KUKA KRL program: MyProgram_307().src

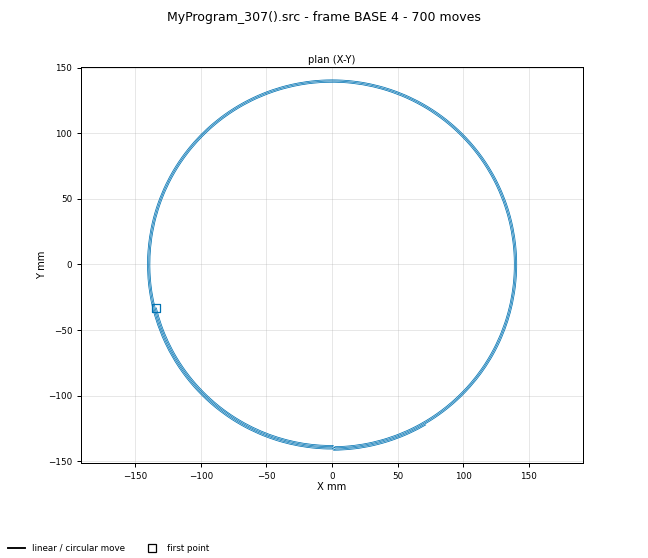
[picture p0: tool path of MyProgram_307().src in frame BASE 4, 700 of 700 moves have a stored position in this frame; points joined in program order, loops and branches not executed]
&ACCESS RVP
&REL 1
&PARAM TEMPLATE = C:\KRC\Roboter\Template\vorgabe
&PARAM EDITMASK = *
DEF MyProgram_307()
; ---- Setting reference (Base) ----
$BASE = BASE_DATA[4]

; --------------------------
; ---- Setting tool (TCP) ----
$TOOL = TOOL_DATA[3]
; --------------------------

$VEL.CP = VEL_APROX_PRINT
Startdeposition()
$VEL.CP = VEL_PRINT
LIN {X -133.9454,Y -33.1389,Z 181,A -162.6013,B 4.9215,C 0.2681,E1 4.7737,E2 255.2334} C_DIS
LIN {X -133.0835,Y -36.4443,Z 181,A -161.1714,B 4.9213,C 0.2719,E1 4.7748,E2 253.8028} C_DIS
LIN {X -132.1601,Y -39.6627,Z 181,A -159.6112,B 4.9212,C 0.2743,E1 4.776,E2 252.2216} C_DIS
LIN {X -131.0021,Y -43.3286,Z 181,A -158.3104,B 4.9208,C 0.281,E1 4.7771,E2 250.9596} C_DIS
LIN {X -130.0909,Y -45.9991,Z 181,A -156.8889,B 4.9208,C 0.2821,E1 4.7784,E2 249.5068} C_DIS
LIN {X -128.9156,Y -49.197,Z 181,A -155.4326,B 4.9206,C 0.2855,E1 4.7799,E2 248.0458} C_DIS
LIN {X -127.6547,Y -52.3816,Z 181,A -153.8465,B 4.9204,C 0.2878,E1 4.7816,E2 246.4393} C_DIS
LIN {X -126.1973,Y -55.7978,Z 181,A -152.4467,B 4.9201,C 0.293,E1 4.7831,E2 245.0586} C_DIS
LIN {X -124.8363,Y -58.7818,Z 181,A -150.8642,B 4.9201,C 0.2946,E1 4.785,E2 243.4483} C_DIS
LIN {X -123.2121,Y -62.1117,Z 181,A -149.5083,B 4.9197,C 0.3,E1 4.7866,E2 242.1167} C_DIS
LIN {X -121.7573,Y -64.9208,Z 181,A -148.0396,B 4.9196,C 0.3019,E1 4.7886,E2 240.6286} C_DIS
LIN {X -120.0477,Y -68.0299,Z 181,A -146.5532,B 4.9194,C 0.3054,E1 4.7906,E2 239.1411} C_DIS
LIN {X -118.3012,Y -71.0238,Z 181,A -144.9881,B 4.9192,C 0.3078,E1 4.7929,E2 237.5603} C_DIS
LIN {X -115.9729,Y -74.7653,Z 181,A -143.1731,B 4.9189,C 0.3122,E1 4.7956,E2 235.7479} C_DIS
LIN {X -113.6464,Y -78.2554,Z 181,A -141.3172,B 4.9188,C 0.3153,E1 4.7985,E2 233.8778} C_DIS
LIN {X -111.4357,Y -81.3732,Z 181,A -139.7753,B 4.9185,C 0.3192,E1 4.801,E2 232.3423} C_DIS
LIN {X -108.9308,Y -84.6964,Z 181,A -137.9766,B 4.9183,C 0.3224,E1 4.8041,E2 230.5349} C_DIS
LIN {X -106.5606,Y -87.6608,Z 181,A -136.3073,B 4.9181,C 0.325,E1 4.807,E2 228.8539} C_DIS
LIN {X -103.6734,Y -91.0571,Z 181,A -134.4884,B 4.9178,C 0.3291,E1 4.8103,E2 227.0397} C_DIS
LIN {X -101.2506,Y -93.7435,Z 181,A -132.8508,B 4.9178,C 0.3309,E1 4.8135,E2 225.3848} C_DIS
LIN {X -98.1988,Y -96.9358,Z 181,A -131.0819,B 4.9174,C 0.3351,E1 4.8169,E2 223.6247} C_DIS
LIN {X -95.6221,Y -99.4784,Z 181,A -129.5752,B 4.9172,C 0.338,E1 4.8199,E2 222.1178} C_DIS
LIN {X -93.0512,Y -101.8874,Z 181,A -127.9603,B 4.9172,C 0.3393,E1 4.8233,E2 220.4833} C_DIS
LIN {X -89.6728,Y -104.8729,Z 181,A -126.0813,B 4.9169,C 0.3425,E1 4.8272,E2 218.6037} C_DIS
LIN {X -86.2779,Y -107.6833,Z 181,A -124.1787,B 4.9168,C 0.345,E1 4.8314,E2 216.6918} C_DIS
LIN {X -82.7629,Y -110.4077,Z 181,A -122.4231,B 4.9165,C 0.3489,E1 4.8352,E2 214.9482} C_DIS
LIN {X -79.8947,Y -112.5007,Z 181,A -120.9123,B 4.9163,C 0.3508,E1 4.8387,E2 213.4328} C_DIS
LIN {X -76.4419,Y -114.8741,Z 181,A -119.086,B 4.9163,C 0.3526,E1 4.8429,E2 211.5952} C_DIS
LIN {X -73.276,Y -116.9196,Z 181,A -117.5586,B 4.916,C 0.3552,E1 4.8465,E2 210.0728} C_DIS
LIN {X -70.2278,Y -118.7753,Z 181,A -115.9776,B 4.916,C 0.3562,E1 4.8503,E2 208.4787} C_DIS
LIN {X -66.4176,Y -120.9472,Z 181,A -114.1055,B 4.9158,C 0.3581,E1 4.8549,E2 206.5998} C_DIS
LIN {X -63.2919,Y -122.6113,Z 181,A -112.7723,B 4.9156,C 0.3612,E1 4.8582,E2 205.2846} C_DIS
LIN {X -60.2633,Y -124.1285,Z 181,A -111.1759,B 4.9156,C 0.3609,E1 4.8622,E2 203.663} C_DIS
LIN {X -56.7836,Y -125.7564,Z 181,A -109.8433,B 4.9153,C 0.3653,E1 4.8655,E2 202.3647} C_DIS
LIN {X -53.8827,Y -127.0278,Z 181,A -108.3761,B 4.9153,C 0.365,E1 4.8694,E2 200.8775} C_DIS
LIN {X -50.3865,Y -128.4531,Z 181,A -106.7907,B 4.9153,C 0.3663,E1 4.8735,E2 199.2895} C_DIS
LIN {X -47.5135,Y -129.5449,Z 181,A -105.5083,B 4.9151,C 0.3674,E1 4.8768,E2 198.0061} C_DIS
LIN {X -44.31,Y -130.6753,Z 181,A -104.1213,B 4.9151,C 0.3688,E1 4.8805,E2 196.6219} C_DIS
LIN {X -41.1844,Y -131.6944,Z 181,A -102.7141,B 4.915,C 0.3694,E1 4.8842,E2 195.2089} C_DIS
LIN {X -37.5841,Y -132.7648,Z 181,A -101.2065,B 4.9149,C 0.3709,E1 4.8883,E2 193.7077} C_DIS
LIN {X -34.6619,Y -133.5589,Z 181,A -99.8819,B 4.9149,C 0.3709,E1 4.8919,E2 192.374} C_DIS
LIN {X -31.53,Y -134.3332,Z 181,A -98.5369,B 4.9149,C 0.3717,E1 4.8955,E2 191.0279} C_DIS
LIN {X -28.3156,Y -135.0474,Z 181,A -97.0137,B 4.9149,C 0.3706,E1 4.8998,E2 189.4836} C_DIS
LIN {X -25.022,Y -135.6957,Z 181,A -95.7674,B 4.9147,C 0.3728,E1 4.9031,E2 188.2564} C_DIS
LIN {X -21.8242,Y -136.2466,Z 181,A -94.4178,B 4.9147,C 0.3732,E1 4.9068,E2 186.9061} C_DIS
LIN {X -18.6385,Y -136.7188,Z 181,A -93.1102,B 4.9147,C 0.3739,E1 4.9104,E2 185.6019} C_DIS
LIN {X -15.2679,Y -137.1353,Z 181,A -91.5885,B 4.9147,C 0.3729,E1 4.9147,E2 184.0648} C_DIS
LIN {X -11.9688,Y -137.4621,Z 181,A -90.4499,B 4.9145,C 0.3758,E1 4.9178,E2 182.9572} C_DIS
LIN {X -9.1803,Y -137.6777,Z 181,A -89.1322,B 4.9146,C 0.3741,E1 4.9215,E2 181.6184} C_DIS
LIN {X -6.0683,Y -137.85,Z 181,A -87.8401,B 4.9146,C 0.3741,E1 4.9251,E2 180.326} C_DIS
LIN {X -3.0627,Y -137.9499,Z 181,A -86.4861,B 4.9147,C 0.3729,E1 4.929,E2 178.9576} C_DIS
LIN {X 0.9801,Y -137.9766,Z 181,A -85.0086,B 4.9146,C 0.375,E1 4.933,E2 177.5057} C_DIS
Enddeposition()
LIN {X 0.9801,Y -137.9766,Z 181,A -85.0086,B 4.9146,C 0.375,E1 4.933,E2 177.5057} C_DIS
Startdeposition()
$VEL.CP = VEL_PRINT
LIN {X 0.4944,Y -138.8836,Z 181,A -85.7347,B 4.875,C 0.383,E1 4.8918,E2 178.3446} C_DIS
LIN {X -3.4627,Y -138.8415,Z 181,A -87.1326,B 4.8752,C 0.3804,E1 4.888,E2 179.7123} C_DIS
LIN {X -6.7652,Y -138.7194,Z 181,A -88.6236,B 4.8752,C 0.3819,E1 4.8838,E2 181.2208} C_DIS
LIN {X -9.6172,Y -138.5516,Z 181,A -89.9061,B 4.875,C 0.383,E1 4.8802,E2 182.5175} C_DIS
LIN {X -13.3672,Y -138.2393,Z 181,A -91.4197,B 4.875,C 0.3824,E1 4.876,E2 184.0265} C_DIS
LIN {X -17.5636,Y -137.7698,Z 181,A -93.0747,B 4.8752,C 0.3811,E1 4.8714,E2 185.6708} C_DIS
LIN {X -21.1736,Y -137.2604,Z 181,A -94.6326,B 4.8752,C 0.3812,E1 4.8671,E2 187.2363} C_DIS
LIN {X -26.796,Y -136.2763,Z 181,A -96.9953,B 4.8752,C 0.3804,E1 4.8606,E2 189.6009} C_DIS
LIN {X -34.4477,Y -134.5442,Z 181,A -100.3956,B 4.8752,C 0.3804,E1 4.8513,E2 193.0236} C_DIS
LIN {X -38.715,Y -133.379,Z 181,A -101.9678,B 4.8755,C 0.3767,E1 4.8471,E2 194.5631} C_DIS
LIN {X -41.235,Y -132.6226,Z 181,A -103.1772,B 4.8755,C 0.3772,E1 4.8439,E2 195.7891} C_DIS
LIN {X -44.9462,Y -131.411,Z 181,A -104.7152,B 4.8756,C 0.3752,E1 4.8398,E2 197.318} C_DIS
LIN {X -48.8191,Y -130.0207,Z 181,A -106.5177,B 4.8756,C 0.3748,E1 4.835,E2 199.1345} C_DIS
LIN {X -51.8681,Y -128.8346,Z 181,A -107.8891,B 4.8757,C 0.3738,E1 4.8315,E2 200.5089} C_DIS
LIN {X -54.7694,Y -127.6288,Z 181,A -109.0264,B 4.8759,C 0.3709,E1 4.8286,E2 201.6256} C_DIS
LIN {X -59.03,Y -125.717,Z 181,A -111.8535,B 4.8754,C 0.3778,E1 4.8211,E2 204.5707} C_DIS
LIN {X -63.9431,Y -123.2899,Z 181,A -113.4971,B 4.8761,C 0.3691,E1 4.8172,E2 206.134} C_DIS
LIN {X -67.9463,Y -121.1302,Z 181,A -115.422,B 4.8762,C 0.3672,E1 4.8125,E2 208.0654} C_DIS
LIN {X -71.7699,Y -118.9046,Z 181,A -117.2904,B 4.8764,C 0.3651,E1 4.808,E2 209.9395} C_DIS
LIN {X -76.6183,Y -115.8401,Z 181,A -119.6162,B 4.8767,C 0.3614,E1 4.8026,E2 212.26} C_DIS
LIN {X -84.2221,Y -110.4349,Z 181,A -123.5852,B 4.877,C 0.3565,E1 4.7935,E2 216.2446} C_DIS
LIN {X -87.516,Y -107.844,Z 181,A -125.375,B 4.8772,C 0.3541,E1 4.7896,E2 218.0422} C_DIS
LIN {X -90.9695,Y -104.9473,Z 181,A -127.3052,B 4.8774,C 0.3515,E1 4.7855,E2 219.9814} C_DIS
LIN {X -94.1981,Y -102.0588,Z 181,A -129.0586,B 4.8776,C 0.3479,E1 4.7819,E2 221.73} C_DIS
LIN {X -97.3086,Y -99.0972,Z 181,A -130.8666,B 4.8779,C 0.3449,E1 4.7782,E2 223.5425} C_DIS
LIN {X -100.4987,Y -95.8605,Z 181,A -132.759,B 4.8781,C 0.3413,E1 4.7745,E2 225.4367} C_DIS
LIN {X -103.3356,Y -92.7954,Z 181,A -134.575,B 4.8783,C 0.3387,E1 4.7711,E2 227.2644} C_DIS
LIN {X -106.3833,Y -89.2849,Z 181,A -136.4902,B 4.8786,C 0.3346,E1 4.7676,E2 229.1787} C_DIS
LIN {X -109.1273,Y -85.9095,Z 181,A -138.2379,B 4.8789,C 0.3304,E1 4.7646,E2 230.9198} C_DIS
LIN {X -111.6331,Y -82.6276,Z 181,A -140.1054,B 4.879,C 0.328,E1 4.7614,E2 232.808} C_DIS
LIN {X -114.241,Y -78.9833,Z 181,A -142.0035,B 4.8793,C 0.3242,E1 4.7583,E2 234.7119} C_DIS
LIN {X -116.2562,Y -75.9861,Z 181,A -143.5562,B 4.8795,C 0.3213,E1 4.7559,E2 236.2723} C_DIS
LIN {X -118.4334,Y -72.5447,Z 181,A -145.232,B 4.8797,C 0.3173,E1 4.7535,E2 237.9468} C_DIS
LIN {X -120.8988,Y -68.358,Z 181,A -147.5502,B 4.8799,C 0.315,E1 4.7502,E2 240.3046} C_DIS
LIN {X -122.5971,Y -65.2626,Z 181,A -148.8178,B 4.8802,C 0.3099,E1 4.7486,E2 241.5473} C_DIS
LIN {X -124.4032,Y -61.7463,Z 181,A -150.4034,B 4.8805,C 0.3055,E1 4.7466,E2 243.1262} C_DIS
LIN {X -125.7912,Y -58.8695,Z 181,A -151.6999,B 4.8807,C 0.302,E1 4.745,E2 244.4194} C_DIS
LIN {X -127.3708,Y -55.3661,Z 181,A -153.2225,B 4.881,C 0.2974,E1 4.7433,E2 245.9331} C_DIS
LIN {X -128.6627,Y -52.2947,Z 181,A -154.5968,B 4.8812,C 0.2938,E1 4.7418,E2 247.3066} C_DIS
LIN {X -129.8975,Y -49.1479,Z 181,A -156.0541,B 4.8814,C 0.2907,E1 4.7403,E2 248.7714} C_DIS
LIN {X -131.4534,Y -44.8238,Z 181,A -158.2954,B 4.8815,C 0.2884,E1 4.7382,E2 251.0561} C_DIS
LIN {X -132.7357,Y -40.8652,Z 181,A -159.9655,B 4.8818,C 0.2834,E1 4.7368,E2 252.7192} C_DIS
LIN {X -133.7465,Y -37.4243,Z 181,A -161.3507,B 4.8821,C 0.2787,E1 4.7357,E2 254.0914} C_DIS
LIN {X -134.4597,Y -34.7807,Z 181,A -162.6813,B 4.8821,C 0.2772,E1 4.7348,E2 255.4472} C_DIS
LIN {X -135.3119,Y -31.2977,Z 181,A -164.1591,B 4.8824,C 0.2731,E1 4.7338,E2 256.9239} C_DIS
LIN {X -135.9929,Y -28.1944,Z 181,A -165.359,B 4.8826,C 0.2686,E1 4.7331,E2 258.1088} C_DIS
LIN {X -136.6755,Y -24.6697,Z 181,A -166.9504,B 4.8828,C 0.2653,E1 4.7323,E2 259.7133} C_DIS
LIN {X -137.2095,Y -21.5023,Z 181,A -168.3304,B 4.883,C 0.2621,E1 4.7317,E2 261.0994} C_DIS
LIN {X -137.6008,Y -18.8473,Z 181,A -169.6654,B 4.883,C 0.2607,E1 4.7312,E2 262.4628} C_DIS
LIN {X -138.0755,Y -14.9645,Z 181,A -171.2559,B 4.8833,C 0.256,E1 4.7306,E2 264.0492} C_DIS
LIN {X -138.4935,Y -10.412,Z 181,A -173.1157,B 4.8836,C 0.2505,E1 4.7302,E2 265.9043} C_DIS
LIN {X -138.7559,Y -5.9941,Z 181,A -175.1528,B 4.8838,C 0.2469,E1 4.7299,E2 267.9671} C_DIS
LIN {X -138.8816,Y -0.8553,Z 181,A -177.5753,B 4.884,C 0.2432,E1 4.7299,E2 270.4261} C_DIS
LIN {X -138.8521,Y 3.0773,Z 181,A -178.8997,B 4.8843,C 0.2363,E1 4.7299,E2 271.7117} C_DIS
LIN {X -138.7439,Y 6.277,Z 181,A 179.7679,B 4.8845,C 0.2327,E1 4.73,E2 273.0446} C_DIS
LIN {X -138.3162,Y 12.5608,Z 181,A 176.8638,B 4.8847,C 0.2276,E1 4.7307,E2 275.9853} C_DIS
LIN {X -137.7408,Y 17.7848,Z 181,A 174.8472,B 4.885,C 0.2204,E1 4.7313,E2 277.9811} C_DIS
LIN {X -137.3589,Y 20.5376,Z 181,A 173.5643,B 4.8851,C 0.2182,E1 4.7318,E2 279.2803} C_DIS
LIN {X -136.7597,Y 24.1988,Z 181,A 172.0031,B 4.8853,C 0.2141,E1 4.7326,E2 280.8441} C_DIS
LIN {X -135.7874,Y 29.1639,Z 181,A 170.1097,B 4.8856,C 0.2068,E1 4.7336,E2 282.7114} C_DIS
LIN {X -135.1804,Y 31.8662,Z 181,A 168.848,B 4.8857,C 0.2046,E1 4.7344,E2 283.9873} C_DIS
LIN {X -134.2777,Y 35.4725,Z 181,A 167.168,B 4.8859,C 0.2015,E1 4.7356,E2 285.6844} C_DIS
LIN {X -133.2631,Y 39.1106,Z 181,A 165.6413,B 4.886,C 0.197,E1 4.7367,E2 287.2058} C_DIS
LIN {X -132.3737,Y 42.0231,Z 181,A 164.275,B 4.8861,C 0.1944,E1 4.7379,E2 288.5848} C_DIS
LIN {X -131.0212,Y 46.0705,Z 181,A 162.3554,B 4.8863,C 0.1909,E1 4.7396,E2 290.523} C_DIS
LIN {X -129.8532,Y 49.2663,Z 181,A 160.5238,B 4.8863,C 0.1905,E1 4.7415,E2 292.4067} C_DIS
LIN {X -128.2055,Y 53.4043,Z 181,A 159.1589,B 4.8866,C 0.182,E1 4.7429,E2 293.7112} C_DIS
LIN {X -126.8991,Y 56.439,Z 181,A 157.8323,B 4.8868,C 0.1782,E1 4.7444,E2 295.0321} C_DIS
LIN {X -125.4412,Y 59.609,Z 181,A 156.2635,B 4.8868,C 0.1755,E1 4.7462,E2 296.6159} C_DIS
LIN {X -124.2073,Y 62.1434,Z 181,A 154.5799,B 4.8868,C 0.1766,E1 4.7484,E2 298.3633} C_DIS
LIN {X -122.152,Y 66.0929,Z 181,A 153.0885,B 4.8871,C 0.1693,E1 4.7503,E2 299.8104} C_DIS
LIN {X -119.9251,Y 70.0521,Z 181,A 151.1744,B 4.8872,C 0.165,E1 4.753,E2 301.7279} C_DIS
LIN {X -117.6653,Y 73.7852,Z 181,A 149.3455,B 4.8874,C 0.1609,E1 4.7557,E2 303.5588} C_DIS
LIN {X -115.2428,Y 77.5143,Z 181,A 147.4169,B 4.8874,C 0.1573,E1 4.7587,E2 305.4975} C_DIS
LIN {X -112.6388,Y 81.2514,Z 181,A 145.5414,B 4.8876,C 0.1529,E1 4.7617,E2 307.3709} C_DIS
LIN {X -109.6966,Y 85.1814,Z 181,A 143.4781,B 4.8877,C 0.1487,E1 4.7652,E2 309.4373} C_DIS
LIN {X -107.1523,Y 88.361,Z 181,A 141.7845,B 4.8879,C 0.1451,E1 4.7682,E2 311.1312} C_DIS
LIN {X -104.6451,Y 91.316,Z 181,A 140.308,B 4.8879,C 0.1407,E1 4.7708,E2 312.5911} C_DIS
LIN {X -102.6132,Y 93.5942,Z 181,A 138.6665,B 4.8879,C 0.1412,E1 4.774,E2 314.279} C_DIS
LIN {X -98.9007,Y 97.5089,Z 181,A 136.5563,B 4.8881,C 0.1358,E1 4.778,E2 316.373} C_DIS
LIN {X -95.8924,Y 100.4682,Z 181,A 134.9128,B 4.8882,C 0.1315,E1 4.7813,E2 318.003} C_DIS
LIN {X -92.6678,Y 103.4499,Z 181,A 132.7945,B 4.8882,C 0.1307,E1 4.7858,E2 320.1578} C_DIS
LIN {X -88.8133,Y 106.7778,Z 181,A 130.7794,B 4.8884,C 0.1262,E1 4.79,E2 322.1606} C_DIS
LIN {X -85.7498,Y 109.2528,Z 181,A 129.1302,B 4.8884,C 0.1235,E1 4.7936,E2 323.8116} C_DIS
LIN {X -82.5228,Y 111.7107,Z 181,A 127.2929,B 4.8884,C 0.1222,E1 4.7978,E2 325.6678} C_DIS
LIN {X -78.2224,Y 114.7635,Z 181,A 125.1824,B 4.8886,C 0.1181,E1 4.8026,E2 327.7686} C_DIS
LIN {X -74.5376,Y 117.1901,Z 181,A 123.3439,B 4.8886,C 0.1156,E1 4.8069,E2 329.6079} C_DIS
LIN {X -70.8603,Y 119.4492,Z 181,A 121.5161,B 4.8886,C 0.1134,E1 4.8113,E2 331.4402} C_DIS
LIN {X -66.8993,Y 121.7123,Z 181,A 119.7049,B 4.8888,C 0.1102,E1 4.8157,E2 333.2412} C_DIS
LIN {X -63.2671,Y 123.6365,Z 181,A 118.1495,B 4.8888,C 0.1068,E1 4.8195,E2 334.7781} C_DIS
LIN {X -61.139,Y 124.7028,Z 181,A 116.618,B 4.8888,C 0.1107,E1 4.8235,E2 336.3765} C_DIS
LIN {X -57.498,Y 126.4254,Z 181,A 115.3336,B 4.8888,C 0.1053,E1 4.8266,E2 337.6135} C_DIS
LIN {X -50.1603,Y 129.5092,Z 181,A 112.0075,B 4.8889,C 0.1023,E1 4.8352,E2 340.9426} C_DIS
LIN {X -46.9783,Y 130.6971,Z 181,A 110.6724,B 4.8889,C 0.1003,E1 4.8387,E2 342.2686} C_DIS
LIN {X -44.2745,Y 131.6382,Z 181,A 109.3595,B 4.8889,C 0.1005,E1 4.8422,E2 343.5971} C_DIS
LIN {X -40.7392,Y 132.7743,Z 181,A 107.8886,B 4.889,C 0.0987,E1 4.8461,E2 345.0594} C_DIS
LIN {X -36.3511,Y 134.0434,Z 181,A 105.8616,B 4.889,C 0.0987,E1 4.8516,E2 347.1029} C_DIS
LIN {X -32.6868,Y 134.9826,Z 181,A 104.5573,B 4.889,C 0.0952,E1 4.8551,E2 348.3746} C_DIS
LIN {X -29.5252,Y 135.7094,Z 181,A 103.2044,B 4.889,C 0.0946,E1 4.8588,E2 349.7285} C_DIS
LIN {X -26.1805,Y 136.394,Z 181,A 101.683,B 4.889,C 0.095,E1 4.863,E2 351.2631} C_DIS
LIN {X -23.3867,Y 136.9018,Z 181,A 100.5739,B 4.8891,C 0.0939,E1 4.866,E2 352.3639} C_DIS
LIN {X -18.7437,Y 137.6151,Z 181,A 98.4444,B 4.8891,C 0.0951,E1 4.8719,E2 354.516} C_DIS
LIN {X -14.9753,Y 138.0743,Z 181,A 96.1048,B 4.8889,C 0.1026,E1 4.8787,E2 356.9492} C_DIS
LIN {X -8.7422,Y 138.6088,Z 181,A 94.3879,B 4.8891,C 0.0933,E1 4.8832,E2 358.5593} C_DIS
LIN {X -5.3578,Y 138.7807,Z 181,A 92.9402,B 4.8891,C 0.0937,E1 4.8872,E2 360.0125} C_DIS
LIN {X -1.1397,Y 138.88,Z 181,A 91.2101,B 4.8891,C 0.0937,E1 4.8921,E2 361.7405} C_DIS
LIN {X 1.7968,Y 138.8735,Z 181,A 90.1301,B 4.8891,C 0.0923,E1 4.895,E2 362.8038} C_DIS
LIN {X 5.3746,Y 138.7801,Z 181,A 88.635,B 4.8891,C 0.0927,E1 4.8992,E2 364.3006} C_DIS
LIN {X 7.8575,Y 138.6633,Z 181,A 87.3994,B 4.8891,C 0.0952,E1 4.9027,E2 365.5618} C_DIS
LIN {X 11.6603,Y 138.3937,Z 181,A 85.9444,B 4.8891,C 0.0944,E1 4.9067,E2 367.0016} C_DIS
LIN {X 15.3454,Y 138.0345,Z 181,A 84.4552,B 4.8891,C 0.0944,E1 4.9109,E2 368.4855} C_DIS
LIN {X 23.4286,Y 136.8948,Z 181,A 81.2082,B 4.8891,C 0.0947,E1 4.9198,E2 371.7167} C_DIS
LIN {X 31.2951,Y 135.3125,Z 181,A 77.7869,B 4.8891,C 0.098,E1 4.9292,E2 375.151} C_DIS
LIN {X 35.2502,Y 134.337,Z 181,A 76.1439,B 4.8891,C 0.0988,E1 4.9336,E2 376.789} C_DIS
LIN {X 38.0632,Y 133.5678,Z 181,A 74.9207,B 4.889,C 0.1001,E1 4.9369,E2 378.0144} C_DIS
LIN {X 41.8152,Y 132.4401,Z 181,A 73.4533,B 4.889,C 0.0997,E1 4.9408,E2 379.463} C_DIS
LIN {X 45.8645,Y 131.0926,Z 181,A 71.5333,B 4.889,C 0.1033,E1 4.9459,E2 381.4025} C_DIS
LIN {X 50.0297,Y 129.56,Z 181,A 69.7647,B 4.8889,C 0.1045,E1 4.9505,E2 383.163} C_DIS
LIN {X 52.8768,Y 128.4258,Z 181,A 68.566,B 4.8889,C 0.1051,E1 4.9536,E2 384.3535} C_DIS
LIN {X 56.2271,Y 126.9938,Z 181,A 67.144,B 4.8889,C 0.1059,E1 4.9572,E2 385.7653} C_DIS
LIN {X 60.9927,Y 124.7749,Z 181,A 64.8954,B 4.8888,C 0.1096,E1 4.963,E2 388.0237} C_DIS
LIN {X 64.6215,Y 122.9337,Z 181,A 63.2427,B 4.8888,C 0.1115,E1 4.967,E2 389.673} C_DIS
LIN {X 68.3111,Y 120.9251,Z 181,A 61.4551,B 4.8887,C 0.1146,E1 4.9714,E2 391.4674} C_DIS
LIN {X 71.9151,Y 118.8168,Z 181,A 59.6705,B 4.8886,C 0.1179,E1 4.9757,E2 393.2596} C_DIS
LIN {X 75.5511,Y 116.5386,Z 181,A 58.1145,B 4.8886,C 0.1181,E1 4.9793,E2 394.7891} C_DIS
LIN {X 81.6596,Y 112.343,Z 181,A 55.002,B 4.8884,C 0.1238,E1 4.9865,E2 397.9087} C_DIS
LIN {X 85.3125,Y 109.595,Z 181,A 53.1419,B 4.8884,C 0.1268,E1 4.9906,E2 399.7658} C_DIS
LIN {X 88.8963,Y 106.7091,Z 181,A 51.2503,B 4.8883,C 0.1302,E1 4.9947,E2 401.6569} C_DIS
LIN {X 92.4054,Y 103.6849,Z 181,A 49.4029,B 4.8882,C 0.133,E1 4.9986,E2 403.4966} C_DIS
LIN {X 95.7081,Y 100.6443,Z 181,A 47.4273,B 4.8881,C 0.1382,E1 5.0026,E2 405.4878} C_DIS
LIN {X 99.4872,Y 96.9106,Z 181,A 45.4732,B 4.8881,C 0.1396,E1 5.0064,E2 407.4128} C_DIS
LIN {X 102.1847,Y 94.0611,Z 181,A 43.8413,B 4.8879,C 0.1432,E1 5.0095,E2 409.0466} C_DIS
LIN {X 105.3046,Y 90.5546,Z 181,A 42.0045,B 4.8879,C 0.146,E1 5.0129,E2 410.8715} C_DIS
LIN {X 107.4021,Y 88.057,Z 181,A 40.562,B 4.8877,C 0.1503,E1 5.0155,E2 412.3266} C_DIS
LIN {X 110.5306,Y 84.097,Z 181,A 38.596,B 4.8877,C 0.1534,E1 5.0188,E2 414.2787} C_DIS
LIN {X 113.1998,Y 80.4683,Z 181,A 36.7609,B 4.8875,C 0.1574,E1 5.0218,E2 416.1114} C_DIS
LIN {X 115.5955,Y 76.9863,Z 181,A 35.0874,B 4.8874,C 0.1606,E1 5.0244,E2 417.7767} C_DIS
LIN {X 117.8647,Y 73.4651,Z 181,A 32.5951,B 4.8869,C 0.175,E1 5.0283,E2 420.3651} C_DIS
LIN {X 121.3088,Y 67.628,Z 181,A 30.6384,B 4.887,C 0.1707,E1 5.0308,E2 422.2182} C_DIS
LIN {X 123.5574,Y 63.4226,Z 181,A 28.9897,B 4.887,C 0.1713,E1 5.0329,E2 423.8274} C_DIS
LIN {X 125.2256,Y 60.0603,Z 181,A 27.1161,B 4.8867,C 0.1797,E1 5.0352,E2 425.7428} C_DIS
LIN {X 127.2538,Y 55.6366,Z 181,A 24.2415,B 4.8861,C 0.1967,E1 5.0386,E2 428.7269} C_DIS
LIN {X 130.3076,Y 48.0531,Z 181,A 21.9685,B 4.8863,C 0.1906,E1 5.0407,E2 430.864} C_DIS
LIN {X 131.6873,Y 44.1272,Z 181,A 20.4175,B 4.8863,C 0.193,E1 5.0421,E2 432.3949} C_DIS
LIN {X 132.7352,Y 40.8669,Z 181,A 19.0565,B 4.8861,C 0.1961,E1 5.0432,E2 433.7501} C_DIS
LIN {X 133.6882,Y 37.6328,Z 181,A 17.7561,B 4.886,C 0.1986,E1 5.0442,E2 435.0397} C_DIS
LIN {X 134.5801,Y 34.3063,Z 181,A 16.3614,B 4.8858,C 0.2022,E1 5.0452,E2 436.432} C_DIS
LIN {X 135.2517,Y 31.5613,Z 181,A 15.0754,B 4.8856,C 0.207,E1 5.046,E2 437.7341} C_DIS
LIN {X 136.5842,Y 25.1796,Z 181,A 12.5906,B 4.8854,C 0.2117,E1 5.0474,E2 440.1945} C_DIS
LIN {X 137.7658,Y 17.5942,Z 181,A 8.9513,B 4.8847,C 0.2272,E1 5.0489,E2 443.8959} C_DIS
LIN {X 138.2931,Y 12.8062,Z 181,A 7.4725,B 4.8848,C 0.2257,E1 5.0493,E2 445.3114} C_DIS
LIN {X 138.5858,Y 9.1154,Z 181,A 6.1341,B 4.8848,C 0.2274,E1 5.0495,E2 446.6267} C_DIS
LIN {X 138.7769,Y 5.4563,Z 181,A 4.5368,B 4.8845,C 0.2329,E1 5.0497,E2 448.2361} C_DIS
LIN {X 138.8787,Y 1.3925,Z 181,A 2.8264,B 4.8842,C 0.2381,E1 5.0498,E2 449.9521} C_DIS
LIN {X 138.8391,Y -3.5486,Z 181,A 1.0016,B 4.8841,C 0.2409,E1 5.0498,E2 451.7509} C_DIS
LIN {X 138.6865,Y -7.4197,Z 181,A -0.641,B 4.8838,C 0.2461,E1 5.0495,E2 453.4004} C_DIS
LIN {X 138.431,Y -11.219,Z 181,A -1.9337,B 4.8838,C 0.2466,E1 5.0493,E2 454.6585} C_DIS
LIN {X 138.0905,Y -14.8251,Z 181,A -3.5008,B 4.8835,C 0.2519,E1 5.0488,E2 456.2362} C_DIS
LIN {X 137.6689,Y -18.3333,Z 181,A -4.728,B 4.8835,C 0.2527,E1 5.0484,E2 457.4347} C_DIS
LIN {X 137.0035,Y -22.7768,Z 181,A -6.6729,B 4.8831,C 0.2593,E1 5.0476,E2 459.3929} C_DIS
LIN {X 136.4329,Y -25.9771,Z 181,A -7.8148,B 4.8831,C 0.2602,E1 5.047,E2 460.5102} C_DIS
LIN {X 135.819,Y -29.0173,Z 181,A -9.3065,B 4.8827,C 0.2668,E1 5.0462,E2 462.0304} C_DIS
LIN {X 135.11,Y -32.1585,Z 181,A -10.6278,B 4.8825,C 0.2704,E1 5.0453,E2 463.3519} C_DIS
LIN {X 133.9712,Y -36.6209,Z 181,A -12.6319,B 4.8822,C 0.2771,E1 5.0439,E2 465.3711} C_DIS
LIN {X 132.384,Y -41.9911,Z 181,A -14.632,B 4.8821,C 0.2791,E1 5.0423,E2 467.3329} C_DIS
LIN {X 131.4752,Y -44.7609,Z 181,A -15.9582,B 4.8818,C 0.2841,E1 5.0411,E2 468.6762} C_DIS
LIN {X 130.0941,Y -48.6232,Z 181,A -17.4787,B 4.8816,C 0.2862,E1 5.0397,E2 470.1758} C_DIS
LIN {X 129.0097,Y -51.4338,Z 181,A -18.7372,B 4.8814,C 0.2898,E1 5.0384,E2 471.4374} C_DIS
LIN {X 127.6641,Y -54.6877,Z 181,A -20.1515,B 4.8812,C 0.2931,E1 5.0369,E2 472.8481} C_DIS
LIN {X 126.1721,Y -58.0459,Z 181,A -21.5854,B 4.8811,C 0.2959,E1 5.0352,E2 474.2725} C_DIS
LIN {X 124.863,Y -60.8141,Z 181,A -22.7598,B 4.8809,C 0.2979,E1 5.0338,E2 475.4366} C_DIS
LIN {X 123.1894,Y -64.1345,Z 181,A -24.3601,B 4.8806,C 0.3028,E1 5.0318,E2 477.0468} C_DIS
LIN {X 121.0072,Y -68.165,Z 181,A -26.2394,B 4.8804,C 0.3074,E1 5.0292,E2 478.9263} C_DIS
LIN {X 118.8168,Y -71.9151,Z 181,A -28.0903,B 4.88,C 0.3127,E1 5.0266,E2 480.7865} C_DIS
LIN {X 116.1817,Y -76.0994,Z 181,A -29.9286,B 4.8799,C 0.3149,E1 5.0238,E2 482.6003} C_DIS
LIN {X 113.8053,Y -79.6095,Z 181,A -31.6792,B 4.8796,C 0.3191,E1 5.0211,E2 484.3526} C_DIS
LIN {X 111.4097,Y -82.9282,Z 181,A -33.1282,B 4.8796,C 0.3198,E1 5.0187,E2 485.7718} C_DIS
LIN {X 109.8516,Y -84.9814,Z 181,A -34.6125,B 4.879,C 0.328,E1 5.0161,E2 487.312} C_DIS
LIN {X 107.6277,Y -87.7809,Z 181,A -35.6175,B 4.8792,C 0.3249,E1 5.0145,E2 488.2569} C_DIS
LIN {X 105.6543,Y -90.1468,Z 181,A -37.0951,B 4.8788,C 0.3306,E1 5.0117,E2 489.7627} C_DIS
LIN {X 102.6332,Y -93.572,Z 181,A -39.1631,B 4.8784,C 0.3372,E1 5.0078,E2 491.8563} C_DIS
LIN {X 100.0797,Y -96.2987,Z 181,A -40.4539,B 4.8784,C 0.3371,E1 5.0054,E2 493.1157} C_DIS
LIN {X 96.8246,Y -99.5705,Z 181,A -42.3048,B 4.8782,C 0.3403,E1 5.0017,E2 494.9613} C_DIS
LIN {X 93.5242,Y -102.6766,Z 181,A -44.0905,B 4.878,C 0.3429,E1 4.9981,E2 496.7376} C_DIS
LIN {X 91.0189,Y -104.9043,Z 181,A -45.5269,B 4.8778,C 0.3464,E1 4.9951,E2 498.1822} C_DIS
LIN {X 87.3953,Y -107.9413,Z 181,A -47.1761,B 4.8778,C 0.3461,E1 4.9916,E2 499.7934} C_DIS
LIN {X 83.4862,Y -110.9918,Z 181,A -49.2192,B 4.8775,C 0.3498,E1 4.9871,E2 501.8379} C_DIS
LIN {X 79.4002,Y -113.951,Z 181,A -51.4179,B 4.8771,C 0.3549,E1 4.982,E2 504.0538} C_DIS
LIN {X 75.7087,Y -116.4362,Z 181,A -53.2184,B 4.8769,C 0.3575,E1 4.9778,E2 505.8511} C_DIS
LIN {X 71.9893,Y -118.7719,Z 181,A -55.1148,B 4.8767,C 0.3615,E1 4.9733,E2 507.7601} C_DIS
LIN {X 66.8547,Y -121.7366,Z 181,A -57.4074,B 4.8765,C 0.3632,E1 4.9678,E2 510.0344} C_DIS
LIN {X 63.578,Y -123.4782,Z 181,A -58.7569,B 4.8765,C 0.3631,E1 4.9645,E2 511.3611} C_DIS
LIN {X 60.2279,Y -125.1455,Z 181,A -60.3713,B 4.8763,C 0.3661,E1 4.9604,E2 512.986} C_DIS
LIN {X 56.9719,Y -126.6607,Z 181,A -61.8128,B 4.8763,C 0.3675,E1 4.9568,E2 514.4233} C_DIS
LIN {X 53.8374,Y -128.0246,Z 181,A -63.2161,B 4.8761,C 0.3691,E1 4.9532,E2 515.8267} C_DIS
LIN {X 50.6593,Y -129.3153,Z 181,A -64.5977,B 4.876,C 0.3704,E1 4.9496,E2 517.2049} C_DIS
LIN {X 47.8314,Y -130.3895,Z 181,A -65.9959,B 4.8757,C 0.3736,E1 4.9459,E2 518.6238} C_DIS
LIN {X 44.2597,Y -131.6432,Z 181,A -67.4206,B 4.8757,C 0.3736,E1 4.9422,E2 520.0315} C_DIS
LIN {X 41.2504,Y -132.6179,Z 181,A -68.5997,B 4.8757,C 0.3733,E1 4.9391,E2 521.195} C_DIS
LIN {X 37.4427,Y -133.7413,Z 181,A -70.0701,B 4.8758,C 0.3727,E1 4.9352,E2 522.6442} C_DIS
LIN {X 34.2504,Y -134.5943,Z 181,A -71.9656,B 4.8752,C 0.3803,E1 4.9299,E2 524.6109} C_DIS
LIN {X 30.91,Y -135.4005,Z 181,A -73.0582,B 4.8754,C 0.3775,E1 4.927,E2 525.6616} C_DIS
LIN {X 27.7361,Y -136.0861,Z 181,A -74.3672,B 4.8754,C 0.3781,E1 4.9234,E2 526.9673} C_DIS
LIN {X 23.3692,Y -136.9047,Z 181,A -76.0893,B 4.8754,C 0.3779,E1 4.9187,E2 528.6759} C_DIS
LIN {X 17.0841,Y -137.8307,Z 181,A -78.9059,B 4.8751,C 0.3816,E1 4.9109,E2 531.5199} C_DIS
LIN {X 13.2866,Y -138.247,Z 181,A -80.3758,B 4.8751,C 0.3811,E1 4.9068,E2 532.9767} C_DIS
LIN {X 9.6364,Y -138.5502,Z 181,A -81.8724,B 4.8751,C 0.3814,E1 4.9026,E2 534.4722} C_DIS
LIN {X 5.8085,Y -138.7632,Z 181,A -83.434,B 4.8751,C 0.3816,E1 4.8983,E2 536.032} C_DIS
LIN {X 2.3643,Y -138.864,Z 181,A -84.9097,B 4.8751,C 0.3825,E1 4.8941,E2 537.5155} C_DIS
LIN {X 2.3643,Y -138.864,Z 181,A -84.9097,B 4.8751,C 0.3825,E1 4.8941,E2 537.5155} C_DIS
Enddeposition()
LIN {X 0.998,Y -139.78,Z 181,A -84.9749,B 4.8345,C 0.3788,E1 4.8533,E2 537.5584} C_DIS
Startdeposition()
$VEL.CP = VEL_PRINT
LIN {X 4.0371,Y -139.7283,Z 181,A -83.5714,B 4.8346,C 0.3767,E1 4.8572,E2 536.1332} C_DIS
LIN {X 7.3998,Y -139.591,Z 181,A -82.163,B 4.8346,C 0.376,E1 4.8612,E2 534.7203} C_DIS
LIN {X 11.0635,Y -139.3497,Z 181,A -80.5381,B 4.8348,C 0.3741,E1 4.8658,E2 533.0784} C_DIS
LIN {X 14.9873,Y -138.9806,Z 181,A -79.0366,B 4.8348,C 0.3748,E1 4.8699,E2 531.5913} C_DIS
LIN {X 19.0382,Y -138.4856,Z 181,A -77.0101,B 4.8352,C 0.3698,E1 4.8756,E2 529.5162} C_DIS
LIN {X 22.7089,Y -137.9297,Z 181,A -76.0761,B 4.8347,C 0.3759,E1 4.878,E2 528.6605} C_DIS
LIN {X 28.1751,Y -136.9177,Z 181,A -74.0311,B 4.8346,C 0.3773,E1 4.8836,E2 526.6455} C_DIS
LIN {X 31.0752,Y -136.2883,Z 181,A -71.95,B 4.8355,C 0.3659,E1 4.8895,E2 524.4473} C_DIS
LIN {X 35.3263,Y -135.2506,Z 181,A -70.5785,B 4.8352,C 0.3696,E1 4.8931,E2 523.1318} C_DIS
LIN {X 40.0072,Y -133.9408,Z 181,A -68.6784,B 4.8352,C 0.3689,E1 4.8982,E2 521.2429} C_DIS
LIN {X 42.7538,Y -133.0876,Z 181,A -67.4647,B 4.8354,C 0.3673,E1 4.9014,E2 520.0236} C_DIS
LIN {X 46.2041,Y -131.9299,Z 181,A -65.9853,B 4.8354,C 0.3659,E1 4.9053,E2 518.5449} C_DIS
LIN {X 49.7703,Y -130.628,Z 181,A -64.33,B 4.8357,C 0.3629,E1 4.9097,E2 516.8751} C_DIS
LIN {X 53.8319,Y -129.0048,Z 181,A -62.6406,B 4.8357,C 0.3621,E1 4.914,E2 515.1983} C_DIS
LIN {X 57.2773,Y -127.5126,Z 181,A -61.1762,B 4.8358,C 0.3611,E1 4.9177,E2 513.7429} C_DIS
LIN {X 60.4029,Y -126.062,Z 181,A -59.7691,B 4.836,C 0.3593,E1 4.9213,E2 512.3354} C_DIS
LIN {X 63.5714,Y -124.4942,Z 181,A -58.3184,B 4.8361,C 0.3573,E1 4.9249,E2 510.8833} C_DIS
LIN {X 67.2431,Y -122.5527,Z 181,A -56.0459,B 4.8368,C 0.3474,E1 4.9307,E2 508.5326} C_DIS
LIN {X 71.8447,Y -119.9129,Z 181,A -54.694,B 4.8363,C 0.3548,E1 4.9337,E2 507.29} C_DIS
LIN {X 76.0217,Y -117.3089,Z 181,A -52.6076,B 4.8366,C 0.3506,E1 4.9386,E2 505.1928} C_DIS
LIN {X 79.3106,Y -115.1111,Z 181,A -50.6096,B 4.8371,C 0.3429,E1 4.9434,E2 503.1429} C_DIS
LIN {X 82.364,Y -112.9467,Z 181,A -49.4544,B 4.837,C 0.3452,E1 4.9459,E2 502.0375} C_DIS
LIN {X 85.7552,Y -110.3936,Z 181,A -47.6526,B 4.8373,C 0.3413,E1 4.9499,E2 500.2259} C_DIS
LIN {X 89.1806,Y -107.6452,Z 181,A -45.8695,B 4.8375,C 0.3381,E1 4.9537,E2 498.4435} C_DIS
LIN {X 92.0347,Y -105.2156,Z 181,A -44.4193,B 4.8376,C 0.3363,E1 4.9568,E2 497.0036} C_DIS
LIN {X 95.2741,Y -102.2913,Z 181,A -42.6315,B 4.8379,C 0.3327,E1 4.9605,E2 495.2145} C_DIS
LIN {X 98.6584,Y -99.0314,Z 181,A -40.7627,B 4.8381,C 0.3295,E1 4.9642,E2 493.3517} C_DIS
LIN {X 101.7542,Y -95.8476,Z 181,A -39.1497,B 4.8381,C 0.3285,E1 4.9672,E2 491.7647} C_DIS
LIN {X 104.8141,Y -92.4916,Z 181,A -37.244,B 4.8385,C 0.3238,E1 4.9708,E2 489.8516} C_DIS
LIN {X 107.3241,Y -89.5675,Z 181,A -35.6059,B 4.8387,C 0.3195,E1 4.9738,E2 488.2043} C_DIS
LIN {X 112.2788,Y -83.2719,Z 181,A -32.6403,B 4.839,C 0.3163,E1 4.9788,E2 485.2784} C_DIS
LIN {X 114.026,Y -80.8632,Z 181,A -31.4278,B 4.8391,C 0.3136,E1 4.9808,E2 484.0659} C_DIS
LIN {X 115.9162,Y -78.1293,Z 181,A -29.872,B 4.8395,C 0.3076,E1 4.9833,E2 482.483} C_DIS
LIN {X 119.6744,Y -72.2407,Z 181,A -27.1201,B 4.8399,C 0.3021,E1 4.9874,E2 479.7436} C_DIS
LIN {X 121.7339,Y -68.7138,Z 181,A -25.4328,B 4.8401,C 0.2978,E1 4.9897,E2 478.053} C_DIS
LIN {X 123.81,Y -64.8937,Z 181,A -23.7704,B 4.8403,C 0.2949,E1 4.9919,E2 476.4049} C_DIS
LIN {X 125.6096,Y -61.3405,Z 181,A -22.2333,B 4.8405,C 0.292,E1 4.9938,E2 474.8791} C_DIS
LIN {X 126.9674,Y -58.4759,Z 181,A -20.9397,B 4.8407,C 0.2887,E1 4.9953,E2 473.5852} C_DIS
LIN {X 128.4557,Y -55.1306,Z 181,A -19.4651,B 4.8409,C 0.2851,E1 4.9969,E2 472.1127} C_DIS
LIN {X 129.7721,Y -51.9562,Z 181,A -18.1433,B 4.841,C 0.2826,E1 4.9983,E2 470.8012} C_DIS
LIN {X 130.9402,Y -48.9368,Z 181,A -16.8021,B 4.8413,C 0.2788,E1 4.9996,E2 469.457} C_DIS
LIN {X 132.1026,Y -45.706,Z 181,A -15.4003,B 4.8415,C 0.2751,E1 5.0009,E2 468.0547} C_DIS
LIN {X 133.2118,Y -42.3651,Z 181,A -13.4173,B 4.8421,C 0.2635,E1 5.0027,E2 465.9987} C_DIS
LIN {X 134.7611,Y -37.1466,Z 181,A -11.9506,B 4.8418,C 0.2683,E1 5.0037,E2 464.6317} C_DIS
LIN {X 135.9013,Y -32.7261,Z 181,A -10.0545,B 4.8422,C 0.2627,E1 5.005,E2 462.7308} C_DIS
LIN {X 136.7045,Y -29.192,Z 181,A -8.5998,B 4.8424,C 0.259,E1 5.0059,E2 461.2789} C_DIS
LIN {X 137.971,Y -22.4616,Z 181,A -5.931,B 4.8427,C 0.2531,E1 5.0072,E2 458.6262} C_DIS
LIN {X 138.3457,Y -20.0182,Z 181,A -4.9156,B 4.8428,C 0.2502,E1 5.0076,E2 457.6096} C_DIS
LIN {X 138.827,Y -16.3503,Z 181,A -3.4586,B 4.843,C 0.2468,E1 5.0081,E2 456.1593} C_DIS
LIN {X 139.2039,Y -12.7615,Z 181,A -2.0099,B 4.8432,C 0.243,E1 5.0085,E2 454.7135} C_DIS
LIN {X 139.5171,Y -8.6743,Z 181,A -0.3108,B 4.8434,C 0.238,E1 5.0088,E2 453.0106} C_DIS
LIN {X 139.7249,Y -4.1566,Z 181,A 1.4575,B 4.8436,C 0.2339,E1 5.009,E2 451.2521} C_DIS
LIN {X 139.7866,Y -0.3566,Z 181,A 3.0491,B 4.8439,C 0.229,E1 5.009,E2 449.6549} C_DIS
LIN {X 139.7315,Y 3.9212,Z 181,A 4.6513,B 4.8439,C 0.2262,E1 5.009,E2 448.0713} C_DIS
LIN {X 139.5721,Y 7.775,Z 181,A 6.3037,B 4.8442,C 0.2207,E1 5.0087,E2 446.4085} C_DIS
LIN {X 139.2873,Y 11.8023,Z 181,A 7.7617,B 4.8443,C 0.2188,E1 5.0084,E2 444.9749} C_DIS
LIN {X 138.9409,Y 15.3559,Z 181,A 9.3083,B 4.8446,C 0.2135,E1 5.008,E2 443.4165} C_DIS
LIN {X 137.8278,Y 23.3194,Z 181,A 11.9915,B 4.8446,C 0.2129,E1 5.007,E2 440.8109} C_DIS
LIN {X 136.9118,Y 28.2038,Z 181,A 14.5414,B 4.8451,C 0.2,E1 5.0056,E2 438.1931} C_DIS
LIN {X 136.0741,Y 32.0092,Z 181,A 15.9053,B 4.8451,C 0.1988,E1 5.0047,E2 436.8587} C_DIS
LIN {X 134.9382,Y 36.4979,Z 181,A 17.7483,B 4.8454,C 0.1944,E1 5.0035,E2 435.0216} C_DIS
LIN {X 134.0855,Y 39.5131,Z 181,A 19.0507,B 4.8455,C 0.1906,E1 5.0024,E2 433.7162} C_DIS
LIN {X 133.077,Y 42.7868,Z 181,A 20.4016,B 4.8456,C 0.1876,E1 5.0013,E2 432.3713} C_DIS
LIN {X 131.9647,Y 46.1038,Z 181,A 21.8349,B 4.8458,C 0.1837,E1 5,E2 430.9374} C_DIS
LIN {X 130.1008,Y 51.1275,Z 181,A 24.3727,B 4.8462,C 0.1731,E1 4.9974,E2 428.3541} C_DIS
LIN {X 128.4815,Y 55.0711,Z 181,A 25.4812,B 4.846,C 0.1774,E1 4.9963,E2 427.3275} C_DIS
LIN {X 126.7172,Y 59.017,Z 181,A 27.3705,B 4.8462,C 0.1712,E1 4.9941,E2 425.4222} C_DIS
LIN {X 125.1202,Y 62.3324,Z 181,A 28.8465,B 4.8464,C 0.1678,E1 4.9923,E2 423.9497} C_DIS
LIN {X 123.3489,Y 65.7716,Z 181,A 30.4993,B 4.8465,C 0.1629,E1 4.9901,E2 422.2876} C_DIS
LIN {X 120.9205,Y 70.134,Z 181,A 32.7669,B 4.8468,C 0.1548,E1 4.987,E2 419.9905} C_DIS
LIN {X 118.8345,Y 73.6146,Z 181,A 34.1017,B 4.8468,C 0.1553,E1 4.9851,E2 418.6976} C_DIS
LIN {X 116.3686,Y 77.4536,Z 181,A 35.9205,B 4.8468,C 0.1515,E1 4.9823,E2 416.8847} C_DIS
LIN {X 113.7843,Y 81.2024,Z 181,A 37.731,B 4.847,C 0.1479,E1 4.9794,E2 415.0807} C_DIS
LIN {X 111.1865,Y 84.7247,Z 181,A 39.501,B 4.8471,C 0.1441,E1 4.9764,E2 413.3132} C_DIS
LIN {X 107.1261,Y 89.8035,Z 181,A 41.983,B 4.8472,C 0.1406,E1 4.9721,E2 410.8539} C_DIS
LIN {X 104.6579,Y 92.6683,Z 181,A 43.5992,B 4.8473,C 0.1364,E1 4.9691,E2 409.2289} C_DIS
LIN {X 101.5104,Y 96.106,Z 181,A 45.4636,B 4.8474,C 0.133,E1 4.9656,E2 407.37} C_DIS
LIN {X 98.358,Y 99.3299,Z 181,A 47.8158,B 4.8477,C 0.1227,E1 4.9608,E2 404.9527} C_DIS
LIN {X 94.5408,Y 102.9695,Z 181,A 49.2528,B 4.8476,C 0.1279,E1 4.958,E2 403.6082} C_DIS
LIN {X 91.7699,Y 105.4466,Z 181,A 50.8668,B 4.8476,C 0.1238,E1 4.9546,E2 401.9824} C_DIS
LIN {X 88.1697,Y 108.4754,Z 181,A 52.7603,B 4.8478,C 0.1207,E1 4.9506,E2 400.0932} C_DIS
LIN {X 84.6719,Y 111.2269,Z 181,A 54.5717,B 4.8478,C 0.1177,E1 4.9466,E2 398.2833} C_DIS
LIN {X 80.855,Y 114.0318,Z 181,A 56.702,B 4.848,C 0.112,E1 4.9417,E2 396.1288} C_DIS
LIN {X 77.9666,Y 116.0261,Z 181,A 57.6424,B 4.8479,C 0.1159,E1 4.9397,E2 395.2517} C_DIS
LIN {X 73.7547,Y 118.7473,Z 181,A 59.9274,B 4.848,C 0.1098,E1 4.9342,E2 392.9374} C_DIS
LIN {X 69.8074,Y 121.1101,Z 181,A 61.7479,B 4.848,C 0.1079,E1 4.9298,E2 391.1253} C_DIS
LIN {X 65.8663,Y 123.2981,Z 181,A 63.7644,B 4.8482,C 0.1032,E1 4.9248,E2 389.0875} C_DIS
LIN {X 61.6384,Y 125.4626,Z 181,A 65.6772,B 4.8482,C 0.1011,E1 4.9201,E2 387.179} C_DIS
LIN {X 56.7647,Y 127.7419,Z 181,A 67.5827,B 4.8482,C 0.102,E1 4.9153,E2 385.3118} C_DIS
LIN {X 53.7728,Y 129.0295,Z 181,A 68.9692,B 4.8482,C 0.0999,E1 4.9117,E2 383.919} C_DIS
LIN {X 49.921,Y 130.5704,Z 181,A 70.5953,B 4.8482,C 0.0989,E1 4.9075,E2 382.3026} C_DIS
LIN {X 46.2951,Y 131.8984,Z 181,A 72.7007,B 4.8484,C 0.0911,E1 4.9018,E2 380.131} C_DIS
LIN {X 41.7591,Y 133.4053,Z 181,A 74.0915,B 4.8484,C 0.0961,E1 4.8983,E2 378.8128} C_DIS
LIN {X 37.117,Y 134.7694,Z 181,A 76.026,B 4.8484,C 0.095,E1 4.8931,E2 376.8848} C_DIS
LIN {X 34.2378,Y 135.5285,Z 181,A 77.5621,B 4.8484,C 0.0904,E1 4.8889,E2 375.3091} C_DIS
LIN {X 31.0601,Y 136.2918,Z 181,A 78.9382,B 4.8484,C 0.0891,E1 4.8851,E2 373.9287} C_DIS
LIN {X 27.5876,Y 137.0372,Z 181,A 80.0795,B 4.8484,C 0.0918,E1 4.8821,E2 372.8277} C_DIS
LIN {X 23.4052,Y 137.8135,Z 181,A 82.1084,B 4.8484,C 0.0876,E1 4.8764,E2 370.7633} C_DIS
LIN {X 20.0062,Y 138.3475,Z 181,A 83.2845,B 4.8484,C 0.0896,E1 4.8732,E2 369.6172} C_DIS
LIN {X 15.9034,Y 138.8803,Z 181,A 84.8577,B 4.8484,C 0.0902,E1 4.8689,E2 368.0601} C_DIS
LIN {X 12.805,Y 139.1998,Z 181,A 86.1364,B 4.8484,C 0.0898,E1 4.8654,E2 366.7816} C_DIS
LIN {X 9.5678,Y 139.4599,Z 181,A 87.5791,B 4.8484,C 0.0882,E1 4.8613,E2 365.3254} C_DIS
LIN {X 5.5594,Y 139.6759,Z 181,A 89.1355,B 4.8484,C 0.0889,E1 4.857,E2 363.7808} C_DIS
LIN {X 1.9899,Y 139.7727,Z 181,A 90.5628,B 4.8484,C 0.0891,E1 4.853,E2 362.3587} C_DIS
LIN {X -1.968,Y 139.7731,Z 181,A 92.2589,B 4.8484,C 0.0883,E1 4.8483,E2 360.654} C_DIS
LIN {X -5.7313,Y 139.6692,Z 181,A 93.765,B 4.8484,C 0.0887,E1 4.8441,E2 359.1533} C_DIS
LIN {X -10.2185,Y 139.4124,Z 181,A 95.9853,B 4.8485,C 0.085,E1 4.8377,E2 356.8861} C_DIS
LIN {X -14.1892,Y 139.0664,Z 181,A 97.2003,B 4.8485,C 0.0897,E1 4.8345,E2 355.7249} C_DIS
LIN {X -19.2498,Y 138.4555,Z 181,A 100.1179,B 4.8485,C 0.0818,E1 4.8262,E2 352.7035} C_DIS
LIN {X -25.2061,Y 137.4962,Z 181,A 101.6145,B 4.8484,C 0.0929,E1 4.8224,E2 351.3318} C_DIS
LIN {X -29.4035,Y 136.6588,Z 181,A 103.634,B 4.8484,C 0.0911,E1 4.8168,E2 349.28} C_DIS
LIN {X -32.7698,Y 135.8908,Z 181,A 104.9928,B 4.8484,C 0.0925,E1 4.8131,E2 347.9292} C_DIS
LIN {X -36.2597,Y 135.0017,Z 181,A 106.5456,B 4.8484,C 0.0928,E1 4.8089,E2 346.3676} C_DIS
LIN {X -41.126,Y 133.5996,Z 181,A 108.5677,B 4.8484,C 0.0949,E1 4.8035,E2 344.3535} C_DIS
LIN {X -44.5768,Y 132.4886,Z 181,A 110.0707,B 4.8484,C 0.0959,E1 4.7995,E2 342.8493} C_DIS
LIN {X -47.6773,Y 131.4043,Z 181,A 111.4782,B 4.8483,C 0.0966,E1 4.7958,E2 341.435} C_DIS
LIN {X -52.0437,Y 129.7368,Z 181,A 113.7171,B 4.8483,C 0.0954,E1 4.7898,E2 339.1566} C_DIS
LIN {X -55.3264,Y 128.371,Z 181,A 114.5939,B 4.8482,C 0.1024,E1 4.7878,E2 338.3539} C_DIS
LIN {X -58.1282,Y 127.1282,Z 181,A 116.3143,B 4.8482,C 0.0995,E1 4.7832,E2 336.5762} C_DIS
LIN {X -62.0146,Y 125.277,Z 181,A 117.9515,B 4.8482,C 0.1028,E1 4.7792,E2 334.9562} C_DIS
LIN {X -64.9517,Y 123.7795,Z 181,A 119.2588,B 4.8482,C 0.1049,E1 4.7759,E2 333.6554} C_DIS
LIN {X -68.7184,Y 121.7313,Z 181,A 121.1664,B 4.8482,C 0.1059,E1 4.7712,E2 331.7303} C_DIS
LIN {X -72.1109,Y 119.7529,Z 181,A 122.6494,B 4.848,C 0.1093,E1 4.7677,E2 330.2644} C_DIS
LIN {X -75.1891,Y 117.8444,Z 181,A 124.2939,B 4.848,C 0.1101,E1 4.7638,E2 328.6009} C_DIS
LIN {X -78.7712,Y 115.4813,Z 181,A 126.1163,B 4.848,C 0.1122,E1 4.7595,E2 326.7718} C_DIS
LIN {X -84.3871,Y 111.4428,Z 181,A 129.2311,B 4.848,C 0.1144,E1 4.7525,E2 323.6239} C_DIS
LIN {X -87.2651,Y 109.2041,Z 181,A 130.4826,B 4.8478,C 0.1192,E1 4.7498,E2 322.4044} C_DIS
LIN {X -90.5959,Y 106.4568,Z 181,A 132.786,B 4.8478,C 0.1177,E1 4.7447,E2 320.0346} C_DIS
LIN {X -94.2576,Y 103.2293,Z 181,A 134.9204,B 4.8478,C 0.1203,E1 4.7403,E2 317.8848} C_DIS
LIN {X -98.1469,Y 99.5389,Z 181,A 136.4075,B 4.8475,C 0.1307,E1 4.7375,E2 316.4898} C_DIS
LIN {X -100.5315,Y 97.1293,Z 181,A 138.523,B 4.8475,C 0.1274,E1 4.7332,E2 314.2832} C_DIS
LIN {X -103.9641,Y 93.4461,Z 181,A 140.3468,B 4.8475,C 0.1337,E1 4.7299,E2 312.4918} C_DIS
LIN {X -106.2761,Y 90.8084,Z 181,A 141.4018,B 4.8472,C 0.14,E1 4.7281,E2 311.4866} C_DIS
LIN {X -108.55,Y 88.078,Z 181,A 143.0894,B 4.8472,C 0.1412,E1 4.725,E2 309.7709} C_DIS
LIN {X -112.2833,Y 83.2658,Z 181,A 145.4401,B 4.847,C 0.1481,E1 4.7211,E2 307.4408} C_DIS
LIN {X -114.4052,Y 80.3257,Z 181,A 147.1582,B 4.847,C 0.1496,E1 4.7182,E2 305.6945} C_DIS
LIN {X -117.0049,Y 76.49,Z 181,A 149.1348,B 4.8468,C 0.1534,E1 4.7152,E2 303.7098} C_DIS
LIN {X -119.4623,Y 72.5915,Z 181,A 151.0468,B 4.8467,C 0.1578,E1 4.7123,E2 301.7963} C_DIS
LIN {X -121.6837,Y 68.8032,Z 181,A 152.929,B 4.8466,C 0.1615,E1 4.7097,E2 299.9053} C_DIS
LIN {X -124.3513,Y 63.8521,Z 181,A 155.4566,B 4.8464,C 0.1655,E1 4.7064,E2 297.3512} C_DIS
LIN {X -125.8519,Y 60.8426,Z 181,A 156.6461,B 4.8463,C 0.1706,E1 4.705,E2 296.187} C_DIS
LIN {X -127.2351,Y 57.897,Z 181,A 157.9612,B 4.8461,C 0.1742,E1 4.7034,E2 294.8755} C_DIS
LIN {X -128.5586,Y 54.8926,Z 181,A 159.5713,B 4.8461,C 0.1756,E1 4.7016,E2 293.2326} C_DIS
LIN {X -130.7176,Y 49.5311,Z 181,A 161.6452,B 4.8458,C 0.1842,E1 4.6995,E2 291.1985} C_DIS
LIN {X -131.7473,Y 46.7257,Z 181,A 162.9886,B 4.8457,C 0.1865,E1 4.6983,E2 289.841} C_DIS
LIN {X -133.2397,Y 42.2776,Z 181,A 165.0384,B 4.8455,C 0.1907,E1 4.6965,E2 287.7766} C_DIS
LIN {X -134.3047,Y 38.7646,Z 181,A 166.5214,B 4.8453,C 0.195,E1 4.6953,E2 286.2976} C_DIS
LIN {X -135.1135,Y 35.8404,Z 181,A 167.8349,B 4.8453,C 0.1978,E1 4.6943,E2 284.9761} C_DIS
LIN {X -135.9421,Y 32.5569,Z 181,A 169.2483,B 4.8451,C 0.2015,E1 4.6934,E2 283.5606} C_DIS
LIN {X -136.689,Y 29.2635,Z 181,A 171.2467,B 4.8451,C 0.2005,E1 4.6922,E2 281.4841} C_DIS
LIN {X -137.5892,Y 24.6863,Z 181,A 172.6469,B 4.8447,C 0.2099,E1 4.6915,E2 280.1515} C_DIS
LIN {X -138.1379,Y 21.4037,Z 181,A 174.052,B 4.8446,C 0.2134,E1 4.6909,E2 278.7423} C_DIS
LIN {X -138.629,Y 17.952,Z 181,A 175.5541,B 4.8444,C 0.2168,E1 4.6903,E2 277.232} C_DIS
LIN {X -139.3405,Y 11.1721,Z 181,A 179.1231,B 4.8444,C 0.2187,E1 4.6894,E2 273.5646} C_DIS
LIN {X -139.6681,Y 5.7614,Z 181,A -179.2397,B 4.8438,C 0.2296,E1 4.6892,E2 272.0051} C_DIS
LIN {X -139.7771,Y -1.7287,Z 181,A -176.1767,B 4.8434,C 0.2384,E1 4.6892,E2 268.9455} C_DIS
LIN {X -139.5656,Y -7.887,Z 181,A -173.5756,B 4.8431,C 0.245,E1 4.6894,E2 266.3365} C_DIS
LIN {X -139.3511,Y -11.0471,Z 181,A -171.5546,B 4.8431,C 0.2429,E1 4.6899,E2 264.2223} C_DIS
LIN {X -138.8646,Y -16.0352,Z 181,A -169.8581,B 4.8427,C 0.2516,E1 4.6904,E2 262.5739} C_DIS
LIN {X -138.2731,Y -20.5264,Z 181,A -168.1669,B 4.8424,C 0.2581,E1 4.691,E2 260.9057} C_DIS
LIN {X -137.8297,Y -23.308,Z 181,A -166.972,B 4.8422,C 0.261,E1 4.6916,E2 259.7061} C_DIS
LIN {X -137.1375,Y -27.0946,Z 181,A -165.361,B 4.842,C 0.2651,E1 4.6924,E2 258.0919} C_DIS
LIN {X -136.2297,Y -31.3319,Z 181,A -163.5467,B 4.8418,C 0.2697,E1 4.6935,E2 256.2736} C_DIS
LIN {X -135.4842,Y -34.4123,Z 181,A -162.1054,B 4.8416,C 0.2721,E1 4.6945,E2 254.8146} C_DIS
LIN {X -134.5667,Y -37.8419,Z 181,A -160.6872,B 4.8414,C 0.2764,E1 4.6955,E2 253.4021} C_DIS
LIN {X -133.5175,Y -41.3943,Z 181,A -159.1395,B 4.8412,C 0.2802,E1 4.6968,E2 251.8515} C_DIS
LIN {X -132.38,Y -44.903,Z 181,A -157.2445,B 4.8412,C 0.2812,E1 4.6985,E2 249.9071} C_DIS
LIN {X -131.2775,Y -48.029,Z 181,A -155.7461,B 4.841,C 0.2836,E1 4.7,E2 248.391} C_DIS
LIN {X -129.8863,Y -51.6728,Z 181,A -154.5957,B 4.8405,C 0.2915,E1 4.7011,E2 247.3004} C_DIS
LIN {X -128.7325,Y -54.484,Z 181,A -153.1875,B 4.8404,C 0.2934,E1 4.7026,E2 245.8714} C_DIS
LIN {X -126.706,Y -59.0412,Z 181,A -151.1216,B 4.8401,C 0.2984,E1 4.705,E2 243.8037} C_DIS
LIN {X -125.1959,Y -62.1791,Z 181,A -149.6573,B 4.8399,C 0.3017,E1 4.7068,E2 242.3352} C_DIS
LIN {X -123.3932,Y -65.6874,Z 181,A -147.0644,B 4.8401,C 0.2975,E1 4.7104,E2 239.6137} C_DIS
LIN {X -120.0749,Y -71.573,Z 181,A -145.378,B 4.8391,C 0.3133,E1 4.7126,E2 238.0721} C_DIS
LIN {X -118.5882,Y -74.0104,Z 181,A -143.7488,B 4.8392,C 0.3122,E1 4.715,E2 236.3828} C_DIS
LIN {X -116.2666,Y -77.6063,Z 181,A -142.0847,B 4.8389,C 0.317,E1 4.7176,E2 234.7313} C_DIS
LIN {X -113.7395,Y -81.265,Z 181,A -140.2009,B 4.8387,C 0.3207,E1 4.7206,E2 232.8401} C_DIS
LIN {X -111.3865,Y -84.4619,Z 181,A -138.675,B 4.8384,C 0.3251,E1 4.7231,E2 231.328} C_DIS
LIN {X -109.1295,Y -87.3589,Z 181,A -136.9866,B 4.8383,C 0.3268,E1 4.7261,E2 229.6159} C_DIS
LIN {X -106.3452,Y -90.7272,Z 181,A -135.1672,B 4.838,C 0.3303,E1 4.7294,E2 227.7932} C_DIS
LIN {X -103.5133,Y -93.945,Z 181,A -133.39,B 4.8378,C 0.3337,E1 4.7327,E2 226.0137} C_DIS
LIN {X -100.5095,Y -97.152,Z 181,A -131.5217,B 4.8376,C 0.3367,E1 4.7363,E2 224.1368} C_DIS
LIN {X -97.308,Y -100.3585,Z 181,A -129.6213,B 4.8374,C 0.3399,E1 4.7401,E2 222.2311} C_DIS
LIN {X -93.8353,Y -103.6128,Z 181,A -127.6583,B 4.8371,C 0.3434,E1 4.7441,E2 220.2668} C_DIS
LIN {X -90.5394,Y -106.5048,Z 181,A -125.8089,B 4.8369,C 0.3461,E1 4.748,E2 218.4107} C_DIS
LIN {X -86.9869,Y -109.4256,Z 181,A -123.9169,B 4.8367,C 0.3492,E1 4.7522,E2 216.518} C_DIS
LIN {X -82.393,Y -112.9241,Z 181,A -121.173,B 4.8367,C 0.3494,E1 4.7584,E2 213.7238} C_DIS
LIN {X -79.1415,Y -115.2271,Z 181,A -119.8455,B 4.8363,C 0.3548,E1 4.7614,E2 212.4374} C_DIS
LIN {X -75.4395,Y -117.6842,Z 181,A -118.0497,B 4.8361,C 0.3577,E1 4.7656,E2 210.6449} C_DIS
LIN {X -72.066,Y -119.78,Z 181,A -116.368,B 4.8359,C 0.3594,E1 4.7696,E2 208.9561} C_DIS
LIN {X -68.4235,Y -121.8971,Z 181,A -114.5429,B 4.8359,C 0.3607,E1 4.7741,E2 207.1177} C_DIS
LIN {X -64.5109,Y -124.011,Z 181,A -112.4287,B 4.8359,C 0.36,E1 4.7794,E2 204.9642} C_DIS
LIN {X -60.9782,Y -125.7871,Z 181,A -111.2038,B 4.8355,C 0.3659,E1 4.7823,E2 203.7924} C_DIS
LIN {X -58.5049,Y -126.954,Z 181,A -110.0155,B 4.8355,C 0.3664,E1 4.7854,E2 202.5949} C_DIS
LIN {X -54.8881,Y -128.5606,Z 181,A -108.3492,B 4.8353,C 0.3676,E1 4.7896,E2 200.9225} C_DIS
LIN {X -51.3442,Y -130.0172,Z 181,A -106.7071,B 4.8353,C 0.3683,E1 4.7939,E2 199.2706} C_DIS
LIN {X -44.7912,Y -132.4173,Z 181,A -104.0077,B 4.835,C 0.3724,E1 4.801,E2 196.5922} C_DIS
LIN {X -40.2638,Y -133.8635,Z 181,A -102.0018,B 4.835,C 0.3732,E1 4.8063,E2 194.5782} C_DIS
LIN {X -37.4881,Y -134.6656,Z 181,A -100.4525,B 4.8351,C 0.3701,E1 4.8106,E2 192.9795} C_DIS
LIN {X -34.0611,Y -135.5733,Z 181,A -99.2983,B 4.8348,C 0.3741,E1 4.8137,E2 191.8652} C_DIS
LIN {X -31.0402,Y -136.2963,Z 181,A -97.9785,B 4.8348,C 0.3743,E1 4.8173,E2 190.5387} C_DIS
LIN {X -26.6134,Y -137.2299,Z 181,A -96.0214,B 4.8348,C 0.374,E1 4.8227,E2 188.5672} C_DIS
LIN {X -22.1329,Y -138.025,Z 181,A -94.2466,B 4.8348,C 0.3756,E1 4.8275,E2 186.804} C_DIS
LIN {X -18.276,Y -138.5865,Z 181,A -92.7059,B 4.8346,C 0.3767,E1 4.8318,E2 185.2703} C_DIS
LIN {X -14.7243,Y -139.0089,Z 181,A -91.225,B 4.8346,C 0.3767,E1 4.8359,E2 183.7869} C_DIS
LIN {X -11.5404,Y -139.3094,Z 181,A -89.859,B 4.8346,C 0.3763,E1 4.8397,E2 182.413} C_DIS
LIN {X -7.3791,Y -139.592,Z 181,A -88.1794,B 4.8346,C 0.3767,E1 4.8444,E2 180.7367} C_DIS
LIN {X -3.7871,Y -139.7352,Z 181,A -86.7459,B 4.8346,C 0.3771,E1 4.8484,E2 179.3079} C_DIS
LIN {X 0.1885,Y -139.7876,Z 181,A -85.0113,B 4.8347,C 0.3757,E1 4.8533,E2 177.5584} C_DIS
LIN {X 0.1885,Y -139.7876,Z 181,A -85.0113,B 4.8347,C 0.3757,E1 4.8533,E2 177.5584} C_DIS
Enddeposition()
LIN {X 1.008,Y -140.6831,Z 181,A -84.7734,B 4.6894,C 0.3763,E1 4.7088,E2 177.4066} C_DIS
Startdeposition()
$VEL.CP = VEL_PRINT
LIN {X -3.638,Y -140.6421,Z 181,A -87.1778,B 4.6889,C 0.3822,E1 4.7019,E2 179.881} C_DIS
LIN {X -6.7898,Y -140.5252,Z 181,A -88.4787,B 4.6889,C 0.3824,E1 4.6983,E2 181.1846} C_DIS
LIN {X -11.0196,Y -140.2587,Z 181,A -90.2169,B 4.6889,C 0.3824,E1 4.6934,E2 182.9253} C_DIS
LIN {X -15.0037,Y -139.8864,Z 181,A -91.8385,B 4.6889,C 0.3821,E1 4.6889,E2 184.5464} C_DIS
LIN {X -19.0199,Y -139.3991,Z 181,A -93.6033,B 4.6889,C 0.383,E1 4.684,E2 186.3276} C_DIS
LIN {X -23.0335,Y -138.7904,Z 181,A -95.0006,B 4.6891,C 0.3797,E1 4.6802,E2 187.6911} C_DIS
LIN {X -25.7078,Y -138.3218,Z 181,A -96.281,B 4.6891,C 0.3812,E1 4.6766,E2 188.9954} C_DIS
LIN {X -29.419,Y -137.5786,Z 181,A -97.7833,B 4.6891,C 0.3801,E1 4.6725,E2 190.4929} C_DIS
LIN {X -32.3824,Y -136.9124,Z 181,A -99.0728,B 4.6891,C 0.38,E1 4.669,E2 191.7897} C_DIS
LIN {X -35.5866,Y -136.1151,Z 181,A -100.6647,B 4.689,C 0.3817,E1 4.6646,E2 193.415} C_DIS
LIN {X -38.7993,Y -135.2347,Z 181,A -101.784,B 4.6893,C 0.3784,E1 4.6617,E2 194.503} C_DIS
LIN {X -42.3142,Y -134.1753,Z 181,A -103.1282,B 4.6895,C 0.3758,E1 4.6581,E2 195.8274} C_DIS
LIN {X -47.3725,Y -132.4734,Z 181,A -105.6827,B 4.6893,C 0.3779,E1 4.6512,E2 198.4333} C_DIS
LIN {X -52.1673,Y -130.6599,Z 181,A -107.617,B 4.6896,C 0.3745,E1 4.6463,E2 200.3474} C_DIS
LIN {X -55.9057,Y -129.1037,Z 181,A -109.3444,B 4.6896,C 0.3736,E1 4.6418,E2 202.0855} C_DIS
LIN {X -60.2711,Y -127.125,Z 181,A -111.2211,B 4.6899,C 0.3708,E1 4.6371,E2 203.9524} C_DIS
LIN {X -62.8813,Y -125.8557,Z 181,A -112.6449,B 4.6898,C 0.3718,E1 4.6334,E2 205.4085} C_DIS
LIN {X -66.2152,Y -124.135,Z 181,A -113.9751,B 4.6901,C 0.368,E1 4.6302,E2 206.7126} C_DIS
LIN {X -69.7808,Y -122.1655,Z 181,A -115.6872,B 4.6902,C 0.3664,E1 4.626,E2 208.4319} C_DIS
LIN {X -73.5613,Y -119.927,Z 181,A -117.3142,B 4.6905,C 0.3625,E1 4.6222,E2 210.0373} C_DIS
LIN {X -76.5625,Y -118.0337,Z 181,A -118.9757,B 4.6905,C 0.3625,E1 4.6182,E2 211.7277} C_DIS
LIN {X -80.0647,Y -115.6872,Z 181,A -120.7528,B 4.6907,C 0.3604,E1 4.6141,E2 213.5127} C_DIS
LIN {X -85.7879,Y -111.5095,Z 181,A -123.7178,B 4.691,C 0.3565,E1 4.6074,E2 216.4881} C_DIS
LIN {X -89.4093,Y -108.6274,Z 181,A -125.6376,B 4.6912,C 0.3536,E1 4.6032,E2 218.4124} C_DIS
LIN {X -92.7227,Y -105.8128,Z 181,A -127.3422,B 4.6915,C 0.3499,E1 4.5996,E2 220.108} C_DIS
LIN {X -95.8283,Y -103.0082,Z 181,A -129.1439,B 4.6916,C 0.3476,E1 4.5959,E2 221.9223} C_DIS
LIN {X -99.1607,Y -99.8043,Z 181,A -131.0588,B 4.6919,C 0.3443,E1 4.592,E2 223.8411} C_DIS
LIN {X -102.4221,Y -96.4546,Z 181,A -133.0161,B 4.6921,C 0.341,E1 4.5882,E2 225.8051} C_DIS
LIN {X -105.4117,Y -93.1779,Z 181,A -134.8597,B 4.6924,C 0.3377,E1 4.5848,E2 227.6532} C_DIS
LIN {X -108.3017,Y -89.8026,Z 181,A -136.7061,B 4.6926,C 0.3342,E1 4.5815,E2 229.5039} C_DIS
LIN {X -111.082,Y -86.34,Z 181,A -138.5312,B 4.6929,C 0.3304,E1 4.5783,E2 231.3307} C_DIS
LIN {X -113.9445,Y -82.5253,Z 181,A -140.557,B 4.6931,C 0.3268,E1 4.5749,E2 233.3668} C_DIS
LIN {X -116.6217,Y -78.6967,Z 181,A -142.4692,B 4.6934,C 0.3225,E1 4.5719,E2 235.2797} C_DIS
LIN {X -119.708,Y -73.9183,Z 181,A -144.6198,B 4.6939,C 0.3157,E1 4.5687,E2 237.4075} C_DIS
LIN {X -124.1894,Y -66.1121,Z 181,A -148.6628,B 4.6943,C 0.3099,E1 4.5631,E2 241.4989} C_DIS
LIN {X -126.0176,Y -62.5531,Z 181,A -150.2368,B 4.6946,C 0.3054,E1 4.5611,E2 243.0649} C_DIS
LIN {X -127.3612,Y -59.7743,Z 181,A -151.7613,B 4.6946,C 0.3043,E1 4.5592,E2 244.6239} C_DIS
LIN {X -129.4935,Y -55.0034,Z 181,A -153.8574,B 4.695,C 0.2986,E1 4.5569,E2 246.7147} C_DIS
LIN {X -132.8663,Y -46.258,Z 181,A -157.6154,B 4.6957,C 0.2881,E1 4.5532,E2 250.463} C_DIS
LIN {X -134.0251,Y -42.7846,Z 181,A -159.1547,B 4.6959,C 0.2845,E1 4.5518,E2 252.0077} C_DIS
LIN {X -135.0129,Y -39.5572,Z 181,A -160.5911,B 4.6961,C 0.2813,E1 4.5507,E2 253.4515} C_DIS
LIN {X -136.0234,Y -35.9305,Z 181,A -162.2196,B 4.6963,C 0.2778,E1 4.5495,E2 255.0915} C_DIS
LIN {X -137.034,Y -31.8629,Z 181,A -163.9928,B 4.6965,C 0.2736,E1 4.5483,E2 256.8722} C_DIS
LIN {X -137.8746,Y -27.9977,Z 181,A -165.5702,B 4.6968,C 0.2689,E1 4.5474,E2 258.4443} C_DIS
LIN {X -138.6299,Y -23.9936,Z 181,A -167.4581,B 4.697,C 0.2661,E1 4.5465,E2 260.3608} C_DIS
LIN {X -139.5502,Y -17.8669,Z 181,A -169.7214,B 4.6975,C 0.257,E1 4.5456,E2 262.5887} C_DIS
LIN {X -139.9529,Y -14.3738,Z 181,A -171.7711,B 4.6975,C 0.2576,E1 4.5449,E2 264.7173} C_DIS
LIN {X -140.2917,Y -10.5671,Z 181,A -172.9743,B 4.6978,C 0.2506,E1 4.5447,E2 265.874} C_DIS
LIN {X -140.6695,Y -2.3328,Z 181,A -177.0105,B 4.698,C 0.2461,E1 4.5443,E2 269.995} C_DIS
LIN {X -140.6685,Y 2.3954,Z 181,A -178.4733,B 4.6985,C 0.2372,E1 4.5443,E2 271.3972} C_DIS
LIN {X -140.5425,Y 6.445,Z 181,A 179.7588,B 4.6987,C 0.2334,E1 4.5445,E2 273.179} C_DIS
LIN {X -140.3309,Y 10.0307,Z 181,A 178.3416,B 4.6989,C 0.2289,E1 4.5448,E2 274.5893} C_DIS
LIN {X -139.8556,Y 15.2901,Z 181,A 175.9978,B 4.6991,C 0.2243,E1 4.5454,E2 276.9562} C_DIS
LIN {X -139.1898,Y 20.4907,Z 181,A 173.685,B 4.6993,C 0.2196,E1 4.5463,E2 279.2901} C_DIS
LIN {X -138.0232,Y 27.267,Z 181,A 170.8139,B 4.6997,C 0.2123,E1 4.5477,E2 282.1681} C_DIS
LIN {X -137.0887,Y 31.6235,Z 181,A 169.1476,B 4.7,C 0.2062,E1 4.5487,E2 283.8139} C_DIS
LIN {X -136.0862,Y 35.695,Z 181,A 167.3171,B 4.7001,C 0.2024,E1 4.55,E2 285.6586} C_DIS
LIN {X -135.0447,Y 39.4484,Z 181,A 165.7401,B 4.7003,C 0.198,E1 4.5512,E2 287.2331} C_DIS
LIN {X -134.0345,Y 42.7551,Z 181,A 164.3318,B 4.7005,C 0.1942,E1 4.5524,E2 288.6404} C_DIS
LIN {X -132.8818,Y 46.2134,Z 181,A 162.7309,B 4.7005,C 0.191,E1 4.5538,E2 290.2548} C_DIS
LIN {X -131.3085,Y 50.5128,Z 181,A 160.2958,B 4.7006,C 0.1904,E1 4.5563,E2 292.7606} C_DIS
LIN {X -129.4694,Y 55.0588,Z 181,A 158.8439,B 4.701,C 0.181,E1 4.5578,E2 294.142} C_DIS
LIN {X -128.3022,Y 57.7221,Z 181,A 157.2307,B 4.701,C 0.1812,E1 4.5597,E2 295.8084} C_DIS
LIN {X -126.7113,Y 61.137,Z 181,A 156.173,B 4.7013,C 0.1737,E1 4.5609,E2 296.8045} C_DIS
LIN {X -123.8253,Y 66.7915,Z 181,A 153.2756,B 4.7014,C 0.1696,E1 4.5647,E2 299.7395} C_DIS
LIN {X -121.5619,Y 70.8281,Z 181,A 151.305,B 4.7016,C 0.1656,E1 4.5674,E2 301.7194} C_DIS
LIN {X -119.2694,Y 74.6237,Z 181,A 149.5074,B 4.7017,C 0.1612,E1 4.57,E2 303.5144} C_DIS
LIN {X -116.8295,Y 78.3884,Z 181,A 147.5859,B 4.7018,C 0.1576,E1 4.573,E2 305.4463} C_DIS
LIN {X -114.2973,Y 82.0363,Z 181,A 145.9013,B 4.702,C 0.1524,E1 4.5757,E2 307.1137} C_DIS
LIN {X -111.8628,Y 85.3259,Z 181,A 143.8836,B 4.702,C 0.1514,E1 4.5791,E2 309.1743} C_DIS
LIN {X -108.5858,Y 89.4595,Z 181,A 141.3139,B 4.702,C 0.1501,E1 4.5838,E2 311.7949} C_DIS
LIN {X -105.3044,Y 93.2993,Z 181,A 139.8792,B 4.7024,C 0.1408,E1 4.5863,E2 313.15} C_DIS
LIN {X -100.6052,Y 98.3484,Z 181,A 137.0006,B 4.7025,C 0.1356,E1 4.5918,E2 316.0351} C_DIS
LIN {X -95.7707,Y 103.0619,Z 181,A 134.3545,B 4.7027,C 0.1294,E1 4.5971,E2 318.666} C_DIS
LIN {X -92.9737,Y 105.5917,Z 181,A 132.2531,B 4.7027,C 0.1312,E1 4.6016,E2 320.8372} C_DIS
LIN {X -90.3066,Y 107.8819,Z 181,A 131.0155,B 4.7027,C 0.127,E1 4.6042,E2 322.0494} C_DIS
LIN {X -85.7673,Y 111.5252,Z 181,A 128.3044,B 4.7027,C 0.1258,E1 4.6102,E2 324.8013} C_DIS
LIN {X -82.6796,Y 113.8326,Z 181,A 126.9144,B 4.7029,C 0.1217,E1 4.6133,E2 326.1676} C_DIS
LIN {X -78.4753,Y 116.7714,Z 181,A 124.8524,B 4.7029,C 0.1182,E1 4.618,E2 328.2246} C_DIS
LIN {X -74.5945,Y 119.2875,Z 181,A 123.0343,B 4.7031,C 0.1148,E1 4.6223,E2 330.0332} C_DIS
LIN {X -71.6435,Y 121.0831,Z 181,A 121.488,B 4.7031,C 0.114,E1 4.6261,E2 331.5958} C_DIS
LIN {X -67.6364,Y 123.366,Z 181,A 119.6362,B 4.7031,C 0.1113,E1 4.6306,E2 333.4429} C_DIS
LIN {X -64.0978,Y 125.2388,Z 181,A 118.2036,B 4.7032,C 0.1074,E1 4.634,E2 334.8495} C_DIS
LIN {X -60.1917,Y 127.1629,Z 181,A 116.1403,B 4.7032,C 0.1079,E1 4.6393,E2 336.9479} C_DIS
LIN {X -56.62,Y 128.7947,Z 181,A 114.6637,B 4.7032,C 0.1051,E1 4.643,E2 338.4082} C_DIS
LIN {X -52.9619,Y 130.3396,Z 181,A 112.5752,B 4.7032,C 0.1077,E1 4.6486,E2 340.5542} C_DIS
LIN {X -49.0784,Y 131.8507,Z 181,A 111.305,B 4.7034,C 0.1021,E1 4.6518,E2 341.7701} C_DIS
LIN {X -45.2805,Y 133.2052,Z 181,A 109.4827,B 4.7034,C 0.1024,E1 4.6566,E2 343.6139} C_DIS
LIN {X -41.2214,Y 134.5141,Z 181,A 107.9879,B 4.7034,C 0.0987,E1 4.6605,E2 345.0774} C_DIS
LIN {X -38.7251,Y 135.2565,Z 181,A 106.4809,B 4.7034,C 0.1022,E1 4.6647,E2 346.6395} C_DIS
LIN {X -35.2814,Y 136.1944,Z 181,A 105.2691,B 4.7034,C 0.0989,E1 4.6679,E2 347.8203} C_DIS
LIN {X -30.6961,Y 137.3005,Z 181,A 102.8942,B 4.7034,C 0.1021,E1 4.6745,E2 350.2505} C_DIS
LIN {X -26.184,Y 138.2307,Z 181,A 101.4289,B 4.7034,C 0.0972,E1 4.6784,E2 351.6637} C_DIS
LIN {X -19.5992,Y 139.3171,Z 181,A 98.833,B 4.7035,C 0.095,E1 4.6855,E2 354.2428} C_DIS
LIN {X -15.8777,Y 139.7921,Z 181,A 97.1962,B 4.7035,C 0.0957,E1 4.6901,E2 355.8926} C_DIS
LIN {X -11.9471,Y 140.1806,Z 181,A 95.2704,B 4.7035,C 0.0985,E1 4.6956,E2 357.857} C_DIS
LIN {X -7.8661,Y 140.4709,Z 181,A 93.9744,B 4.7035,C 0.0946,E1 4.6991,E2 359.1063} C_DIS
LIN {X -4.1933,Y 140.6266,Z 181,A 92.4388,B 4.7035,C 0.0949,E1 4.7034,E2 360.6459} C_DIS
LIN {X -0.2046,Y 140.6899,Z 181,A 90.7653,B 4.7035,C 0.0955,E1 4.708,E2 362.3248} C_DIS
LIN {X 3.6887,Y 140.6407,Z 181,A 89.2901,B 4.7035,C 0.0945,E1 4.7121,E2 363.7854} C_DIS
LIN {X 7.8661,Y 140.4709,Z 181,A 87.4851,B 4.7035,C 0.0959,E1 4.7172,E2 365.6027} C_DIS
LIN {X 11.6796,Y 140.2032,Z 181,A 86.061,B 4.7035,C 0.0949,E1 4.7211,E2 367.0095} C_DIS
LIN {X 15.0873,Y 139.8774,Z 181,A 84.6687,B 4.7035,C 0.0954,E1 4.725,E2 368.401} C_DIS
LIN {X 18.7851,Y 139.4299,Z 181,A 82.8333,B 4.7035,C 0.0995,E1 4.7302,E2 370.2757} C_DIS
LIN {X 22.2947,Y 138.9129,Z 181,A 81.6471,B 4.7035,C 0.0974,E1 4.7334,E2 371.4293} C_DIS
LIN {X 25.9292,Y 138.2795,Z 181,A 80.1905,B 4.7035,C 0.0977,E1 4.7373,E2 372.8797} C_DIS
LIN {X 29.5937,Y 137.5409,Z 181,A 78.6861,B 4.7035,C 0.0985,E1 4.7415,E2 374.3813} C_DIS
LIN {X 35.5742,Y 136.1184,Z 181,A 76.1543,B 4.7034,C 0.1007,E1 4.7483,E2 376.9161} C_DIS
LIN {X 39.2935,Y 135.0901,Z 181,A 74.8152,B 4.7034,C 0.0993,E1 4.7519,E2 378.2257} C_DIS
LIN {X 44.4848,Y 133.4704,Z 181,A 72.2889,B 4.7033,C 0.1049,E1 4.7587,E2 380.7907} C_DIS
LIN {X 49.0967,Y 131.8439,Z 181,A 70.4866,B 4.7033,C 0.1047,E1 4.7634,E2 382.5689} C_DIS
LIN {X 52.3271,Y 130.5954,Z 181,A 69.2013,B 4.7033,C 0.1048,E1 4.7667,E2 383.8382} C_DIS
LIN {X 55.0534,Y 129.472,Z 181,A 67.8212,B 4.7033,C 0.1083,E1 4.7703,E2 385.2408} C_DIS
LIN {X 58.6332,Y 127.8888,Z 181,A 66.4648,B 4.7033,C 0.1074,E1 4.7737,E2 386.567} C_DIS
LIN {X 62.284,Y 126.1503,Z 181,A 64.9651,B 4.7033,C 0.1078,E1 4.7774,E2 388.048} C_DIS
LIN {X 64.9376,Y 124.8061,Z 181,A 63.4573,B 4.7031,C 0.1129,E1 4.7812,E2 389.5932} C_DIS
LIN {X 69.0763,Y 122.5653,Z 181,A 61.5948,B 4.7031,C 0.115,E1 4.7858,E2 391.4489} C_DIS
LIN {X 72.7849,Y 120.3998,Z 181,A 59.8286,B 4.703,C 0.1178,E1 4.79,E2 393.2172} C_DIS
LIN {X 76.6415,Y 117.9824,Z 181,A 58.0028,B 4.703,C 0.1204,E1 4.7943,E2 395.0395} C_DIS
LIN {X 80.2845,Y 115.5343,Z 181,A 55.9905,B 4.7028,C 0.126,E1 4.799,E2 397.0801} C_DIS
LIN {X 83.2832,Y 113.3917,Z 181,A 54.7864,B 4.7028,C 0.125,E1 4.8016,E2 398.2471} C_DIS
LIN {X 86.9133,Y 110.6338,Z 181,A 52.968,B 4.7028,C 0.1278,E1 4.8057,E2 400.0608} C_DIS
LIN {X 90.3229,Y 107.8682,Z 181,A 51.1867,B 4.7026,C 0.131,E1 4.8095,E2 401.8414} C_DIS
LIN {X 93.4238,Y 105.1944,Z 181,A 49.335,B 4.7025,C 0.1364,E1 4.8134,E2 403.7166} C_DIS
LIN {X 96.0147,Y 102.8345,Z 181,A 47.8396,B 4.7024,C 0.1401,E1 4.8165,E2 405.2209} C_DIS
LIN {X 98.9771,Y 99.9868,Z 181,A 46.5091,B 4.7024,C 0.1391,E1 4.8191,E2 406.5083} C_DIS
LIN {X 102.1706,Y 96.7212,Z 181,A 44.7502,B 4.7024,C 0.1417,E1 4.8224,E2 408.2548} C_DIS
LIN {X 105.1535,Y 93.47,Z 181,A 42.917,B 4.7022,C 0.146,E1 4.8259,E2 410.0931} C_DIS
LIN {X 108.7592,Y 89.248,Z 181,A 40.6105,B 4.702,C 0.1515,E1 4.83,E2 412.4059} C_DIS
LIN {X 111.9909,Y 85.1584,Z 181,A 38.6512,B 4.702,C 0.1542,E1 4.8334,E2 414.345} C_DIS
LIN {X 114.5981,Y 81.6156,Z 181,A 36.9534,B 4.7018,C 0.1571,E1 4.8361,E2 416.0315} C_DIS
LIN {X 117.103,Y 77.9786,Z 181,A 35.1976,B 4.7018,C 0.1608,E1 4.8389,E2 417.7825} C_DIS
LIN {X 119.5594,Y 74.1577,Z 181,A 33.3916,B 4.7016,C 0.1647,E1 4.8416,E2 419.5835} C_DIS
LIN {X 122.8174,Y 68.6278,Z 181,A 30.8075,B 4.7014,C 0.1707,E1 4.8452,E2 422.1649} C_DIS
LIN {X 125.0011,Y 64.5647,Z 181,A 28.9978,B 4.7012,C 0.1745,E1 4.8475,E2 423.9666} C_DIS
LIN {X 126.7346,Y 61.0882,Z 181,A 27.4979,B 4.7012,C 0.1775,E1 4.8493,E2 425.4566} C_DIS
LIN {X 128.272,Y 57.7897,Z 181,A 26.0572,B 4.701,C 0.1807,E1 4.851,E2 426.8926} C_DIS
LIN {X 129.6888,Y 54.5356,Z 181,A 24.8742,B 4.701,C 0.181,E1 4.8523,E2 428.0426} C_DIS
LIN {X 131.7836,Y 49.2576,Z 181,A 22.5722,B 4.7008,C 0.187,E1 4.8547,E2 430.3445} C_DIS
LIN {X 132.804,Y 46.4378,Z 181,A 21.2522,B 4.7006,C 0.1916,E1 4.8559,E2 431.6779} C_DIS
LIN {X 133.9506,Y 43.0177,Z 181,A 19.8422,B 4.7004,C 0.1947,E1 4.8571,E2 433.0811} C_DIS
LIN {X 134.9659,Y 39.7177,Z 181,A 18.4872,B 4.7004,C 0.1978,E1 4.8582,E2 434.4303} C_DIS
LIN {X 135.9487,Y 36.2105,Z 181,A 17.018,B 4.7001,C 0.2017,E1 4.8593,E2 435.8985} C_DIS
LIN {X 136.9453,Y 32.2458,Z 181,A 15.2914,B 4.6999,C 0.2071,E1 4.8604,E2 437.6342} C_DIS
LIN {X 137.7983,Y 28.3727,Z 181,A 13.7096,B 4.6997,C 0.2112,E1 4.8613,E2 439.2126} C_DIS
LIN {X 138.6579,Y 23.8274,Z 181,A 11.9051,B 4.6995,C 0.2153,E1 4.8622,E2 441.008} C_DIS
LIN {X 139.142,Y 20.8163,Z 181,A 9.9815,B 4.6989,C 0.2282,E1 4.8631,E2 443.0203} C_DIS
LIN {X 139.9457,Y 14.4529,Z 181,A 8.1327,B 4.6991,C 0.2251,E1 4.8636,E2 444.7726} C_DIS
LIN {X 140.3175,Y 10.214,Z 181,A 6.6036,B 4.699,C 0.2272,E1 4.8639,E2 446.2764} C_DIS
LIN {X 140.5326,Y 6.6416,Z 181,A 5.0483,B 4.6987,C 0.2327,E1 4.8642,E2 447.8454} C_DIS
LIN {X 140.6695,Y 2.3376,Z 181,A 3.4326,B 4.6986,C 0.2357,E1 4.8642,E2 449.4444} C_DIS
LIN {X 140.6761,Y -1.9363,Z 181,A 1.7362,B 4.6983,C 0.2401,E1 4.8642,E2 451.1363} C_DIS
LIN {X 140.584,Y -5.4312,Z 181,A 0.3859,B 4.6982,C 0.2431,E1 4.8642,E2 452.4781} C_DIS
LIN {X 140.398,Y -9.0507,Z 181,A -1.0329,B 4.698,C 0.2465,E1 4.8639,E2 453.8905} C_DIS
LIN {X 140.0646,Y -13.2389,Z 181,A -2.7274,B 4.6978,C 0.2511,E1 4.8635,E2 455.5841} C_DIS
LIN {X 139.6517,Y -17.055,Z 181,A -4.254,B 4.6976,C 0.255,E1 4.863,E2 457.1072} C_DIS
LIN {X 139.0613,Y -21.3375,Z 181,A -5.895,B 4.6974,C 0.2583,E1 4.8624,E2 458.7339} C_DIS
LIN {X 137.4771,Y -29.8891,Z 181,A -9.3965,B 4.6969,C 0.2677,E1 4.8605,E2 462.233} C_DIS
LIN {X 135.879,Y -36.4721,Z 181,A -12.3527,B 4.6963,C 0.2781,E1 4.8585,E2 465.2174} C_DIS
LIN {X 134.913,Y -39.8982,Z 181,A -13.7174,B 4.6961,C 0.2809,E1 4.8574,E2 466.5721} C_DIS
LIN {X 133.9544,Y -43.0059,Z 181,A -14.7223,B 4.6961,C 0.2801,E1 4.8566,E2 467.5361} C_DIS
LIN {X 132.8735,Y -46.2373,Z 181,A -16.006,B 4.696,C 0.2824,E1 4.8554,E2 468.8073} C_DIS
LIN {X 131.7673,Y -49.3012,Z 181,A -17.3377,B 4.6958,C 0.286,E1 4.8542,E2 470.1407} C_DIS
LIN {X 130.4928,Y -52.5818,Z 181,A -18.6898,B 4.6956,C 0.2888,E1 4.8528,E2 471.4834} C_DIS
LIN {X 129.2325,Y -55.6078,Z 181,A -20.0679,B 4.6954,C 0.2929,E1 4.8513,E2 472.8683} C_DIS
LIN {X 127.8053,Y -58.8139,Z 181,A -21.4368,B 4.6952,C 0.2958,E1 4.8497,E2 474.2304} C_DIS
LIN {X 126.2765,Y -62.0281,Z 181,A -22.9278,B 4.6949,C 0.3001,E1 4.8479,E2 475.7282} C_DIS
LIN {X 124.4305,Y -65.6529,Z 181,A -24.48,B 4.6947,C 0.3029,E1 4.8459,E2 477.268} C_DIS
LIN {X 122.4213,Y -69.3323,Z 181,A -26.2174,B 4.6944,C 0.3076,E1 4.8436,E2 479.011} C_DIS
LIN {X 120.8243,Y -72.0782,Z 181,A -28.2557,B 4.6935,C 0.3209,E1 4.8405,E2 481.1485} C_DIS
LIN {X 117.2711,Y -77.7267,Z 181,A -30.8294,B 4.6932,C 0.3255,E1 4.8365,E2 483.7056} C_DIS
LIN {X 113.7325,Y -82.8178,Z 181,A -32.685,B 4.6934,C 0.3226,E1 4.8337,E2 485.4752} C_DIS
LIN {X 109.7822,Y -87.9875,Z 181,A -35.2128,B 4.6931,C 0.327,E1 4.8294,E2 487.9891} C_DIS
LIN {X 106.9492,Y -91.4099,Z 181,A -36.9227,B 4.6929,C 0.3297,E1 4.8263,E2 489.6873} C_DIS
LIN {X 104.9803,Y -93.6641,Z 181,A -38.5974,B 4.6923,C 0.3384,E1 4.8231,E2 491.4236} C_DIS
LIN {X 101.6989,Y -97.2168,Z 181,A -40.0521,B 4.6925,C 0.3358,E1 4.8204,E2 492.8118} C_DIS
LIN {X 98.4682,Y -100.4877,Z 181,A -41.8799,B 4.6923,C 0.3391,E1 4.8168,E2 494.6352} C_DIS
LIN {X 95.1237,Y -103.6593,Z 181,A -43.691,B 4.692,C 0.3421,E1 4.8131,E2 496.4391} C_DIS
LIN {X 92.2867,Y -106.1932,Z 181,A -45.232,B 4.6918,C 0.345,E1 4.8099,E2 497.9803} C_DIS
LIN {X 88.8231,Y -109.1067,Z 181,A -47.0105,B 4.6916,C 0.3476,E1 4.8061,E2 499.7516} C_DIS
LIN {X 85.4764,Y -111.7477,Z 181,A -48.722,B 4.6914,C 0.3505,E1 4.8023,E2 501.4613} C_DIS
LIN {X 82.0191,Y -114.3094,Z 181,A -50.8854,B 4.6908,C 0.3588,E1 4.7973,E2 503.6809} C_DIS
LIN {X 78.2818,Y -116.9007,Z 181,A -52.3125,B 4.691,C 0.3566,E1 4.7941,E2 505.0529} C_DIS
LIN {X 75.0706,Y -118.9881,Z 181,A -53.9347,B 4.6907,C 0.3599,E1 4.7903,E2 506.6847} C_DIS
LIN {X 70.0895,Y -121.9894,Z 181,A -56.3768,B 4.6904,C 0.3645,E1 4.7844,E2 509.1384} C_DIS
LIN {X 67.0898,Y -123.6642,Z 181,A -57.4977,B 4.6904,C 0.363,E1 4.7817,E2 510.2232} C_DIS
LIN {X 63.8344,Y -125.3729,Z 181,A -58.9874,B 4.6904,C 0.365,E1 4.778,E2 511.7129} C_DIS
LIN {X 59.8848,Y -127.3095,Z 181,A -60.8159,B 4.6901,C 0.3679,E1 4.7734,E2 513.5478} C_DIS
LIN {X 56.2823,Y -128.9409,Z 181,A -62.3489,B 4.6901,C 0.369,E1 4.7695,E2 515.0715} C_DIS
LIN {X 53.0326,Y -130.3111,Z 181,A -63.7574,B 4.6899,C 0.3703,E1 4.7659,E2 516.4774} C_DIS
LIN {X 49.6313,Y -131.6436,Z 181,A -65.1734,B 4.6899,C 0.3712,E1 4.7622,E2 517.8848} C_DIS
LIN {X 46.3029,Y -132.8508,Z 181,A -66.6774,B 4.6896,C 0.3735,E1 4.7582,E2 519.3981} C_DIS
LIN {X 42.4183,Y -134.1421,Z 181,A -68.211,B 4.6896,C 0.3735,E1 4.7542,E2 520.915} C_DIS
LIN {X 38.2136,Y -135.3997,Z 181,A -70.0347,B 4.6895,C 0.3756,E1 4.7493,E2 522.7447} C_DIS
LIN {X 35.4876,Y -136.1413,Z 181,A -71.8598,B 4.6888,C 0.3845,E1 4.7441,E2 524.6607} C_DIS
LIN {X 30.0061,Y -137.4519,Z 181,A -73.4285,B 4.6893,C 0.3777,E1 4.7401,E2 526.1338} C_DIS
LIN {X 26.6669,Y -138.1384,Z 181,A -74.7906,B 4.6893,C 0.3784,E1 4.7363,E2 527.4933} C_DIS
LIN {X 23.6806,Y -138.6824,Z 181,A -75.9637,B 4.6893,C 0.3784,E1 4.7331,E2 528.6587} C_DIS
LIN {X 17.6037,Y -139.5847,Z 181,A -78.583,B 4.689,C 0.3811,E1 4.7259,E2 531.2952} C_DIS
LIN {X 13.6257,Y -140.0275,Z 181,A -80.1119,B 4.689,C 0.3806,E1 4.7216,E2 532.8114} C_DIS
LIN {X 10.5112,Y -140.2958,Z 181,A -81.477,B 4.689,C 0.3821,E1 4.7178,E2 534.1895} C_DIS
LIN {X 6.5178,Y -140.5388,Z 181,A -83.0297,B 4.689,C 0.3817,E1 4.7135,E2 535.7328} C_DIS
LIN {X 2.5254,Y -140.6663,Z 181,A -84.6973,B 4.689,C 0.3825,E1 4.7088,E2 537.4066} C_DIS
LIN {X 2.5254,Y -140.6663,Z 181,A -84.6973,B 4.689,C 0.3825,E1 4.7088,E2 537.4066} C_DIS
Enddeposition()
LIN {X 1.0182,Y -141.5859,Z 181,A -84.7298,B 4.689,C 0.3787,E1 4.7088,E2 537.3927} C_DIS
Startdeposition()
$VEL.CP = VEL_PRINT
LIN {X 4.7359,Y -141.5141,Z 181,A -83.014,B 4.6893,C 0.376,E1 4.7136,E2 535.6474} C_DIS
LIN {X 8.3503,Y -141.3452,Z 181,A -81.6267,B 4.6893,C 0.3765,E1 4.7174,E2 534.2699} C_DIS
LIN {X 11.7149,Y -141.1058,Z 181,A -80.363,B 4.6893,C 0.3772,E1 4.7209,E2 533.0193} C_DIS
LIN {X 14.6469,Y -140.8324,Z 181,A -79.1942,B 4.6893,C 0.377,E1 4.7241,E2 531.8529} C_DIS
LIN {X 17.7595,Y -140.4743,Z 181,A -77.5864,B 4.6896,C 0.3724,E1 4.7287,E2 530.1979} C_DIS
LIN {X 21.0103,Y -140.0251,Z 181,A -76.6113,B 4.6893,C 0.3758,E1 4.7313,E2 529.2705} C_DIS
LIN {X 24.6207,Y -139.4343,Z 181,A -75.093,B 4.6894,C 0.3745,E1 4.7355,E2 527.7461} C_DIS
LIN {X 27.4319,Y -138.9106,Z 181,A -73.7445,B 4.6897,C 0.3714,E1 4.7393,E2 526.3707} C_DIS
LIN {X 30.7043,Y -138.2242,Z 181,A -72.1316,B 4.69,C 0.3673,E1 4.7438,E2 524.7213} C_DIS
LIN {X 34.6835,Y -137.2773,Z 181,A -70.8613,B 4.6897,C 0.3706,E1 4.7471,E2 523.5027} C_DIS
LIN {X 38.6809,Y -136.206,Z 181,A -69.4037,B 4.6897,C 0.3718,E1 4.7509,E2 522.0738} C_DIS
LIN {X 42.3603,Y -135.1079,Z 181,A -67.6771,B 4.6899,C 0.3682,E1 4.7556,E2 520.3226} C_DIS
LIN {X 46.1774,Y -133.8493,Z 181,A -66.185,B 4.6899,C 0.3682,E1 4.7595,E2 518.8477} C_DIS
LIN {X 49.3989,Y -132.6943,Z 181,A -64.9659,B 4.6899,C 0.3687,E1 4.7626,E2 517.6503} C_DIS
LIN {X 52.515,Y -131.4926,Z 181,A -63.3963,B 4.6902,C 0.3644,E1 4.7668,E2 516.05} C_DIS
LIN {X 55.8773,Y -130.0991,Z 181,A -61.9988,B 4.6902,C 0.3636,E1 4.7704,E2 514.6617} C_DIS
LIN {X 59.1808,Y -128.6298,Z 181,A -60.5982,B 4.6904,C 0.3625,E1 4.7739,E2 513.2685} C_DIS
LIN {X 62.3325,Y -127.1325,Z 181,A -59.0884,B 4.6906,C 0.3594,E1 4.7778,E2 511.7443} C_DIS
LIN {X 65.3162,Y -125.6265,Z 181,A -57.7355,B 4.6907,C 0.3575,E1 4.7811,E2 510.3904} C_DIS
LIN {X 71.3192,Y -122.3203,Z 181,A -54.9619,B 4.6911,C 0.3533,E1 4.7879,E2 507.6147} C_DIS
Enddeposition()
END
